Yaskawa INFORM job: A_NAIHAN_0617_1_PAINT_0.JBI

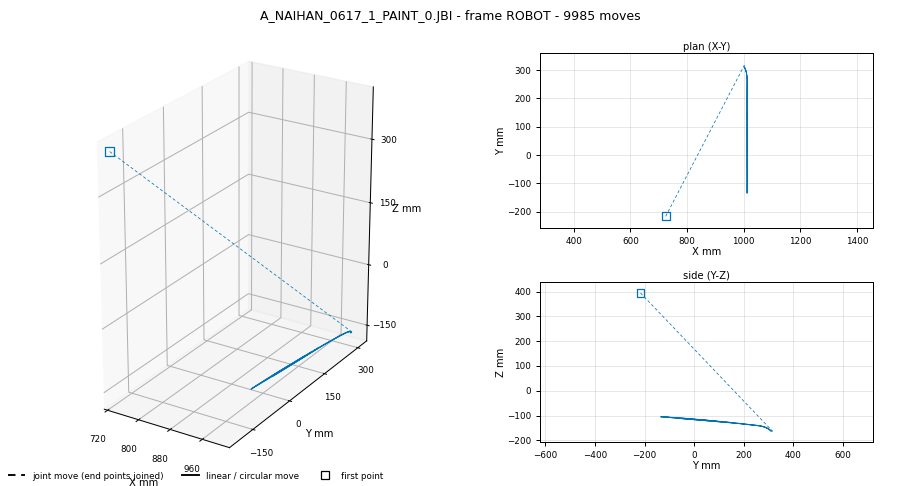
[picture p0: tool path of A_NAIHAN_0617_1_PAINT_0.JBI in frame ROBOT, 9985 of 9985 moves have a stored position in this frame; points joined in program order, loops and branches not executed]
/JOB
//NAME A_NAIHAN_0617_1_PAINT
//POS
///NPOS 9985,0,0,0,0,0
///TOOL 1
///USER 0
///POSTYPE ROBOT
///RECTAN
///RCONF 0,0,0,1,1,0,0,0,0,0,0,0,0,0,0,0,0,0,0,0,0,0,0,0
C00000=724.889,-216.680,394.500,-180.000,-0.000,-0.000
///USER 0
///POSTYPE ROBOT
///RECTAN
///RCONF 0,0,0,0,1,0,0,0,0,0,0,0,0,0,0,0,0,0,0,0,0,0,0,0
C00001=1002.338,316.145,-163.308,164.727,56.498,159.874
///RCONF 0,0,0,0,0,0,0,0,0,0,0,0,0,0,0,0,0,0,0,0,0,0,0,0
C00002=1002.509,311.597,-162.786,164.727,56.498,159.874
C00003=1002.600,311.455,-162.633,164.739,56.513,159.880
C00004=1002.691,311.313,-162.481,164.769,56.519,159.889
C00005=1002.780,311.170,-162.330,164.773,56.536,159.893
C00006=1002.870,311.027,-162.180,164.796,56.545,159.900
C00007=1002.958,310.884,-162.030,164.807,56.560,159.905
///RCONF 0,0,0,0,1,0,0,0,0,0,0,0,0,0,0,0,0,0,0,0,0,0,0,0
C00008=1003.047,310.739,-161.880,164.829,56.569,159.913
C00009=1003.134,310.594,-161.732,164.840,56.583,159.918
C00010=1003.223,310.448,-161.584,164.859,56.594,159.925
C00011=1003.316,310.290,-161.426,164.859,56.615,159.929
C00012=1003.408,310.133,-161.268,164.882,56.624,159.936
C00013=1003.501,309.974,-161.112,164.908,56.633,159.945
C00014=1003.593,309.816,-160.955,164.920,56.648,159.950
C00015=1003.685,309.656,-160.799,164.944,56.657,159.958
C00016=1003.776,309.495,-160.644,164.961,56.670,159.965
C00017=1003.866,309.334,-160.491,164.971,56.686,159.970
C00018=1003.955,309.172,-160.337,164.989,56.698,159.977
C00019=1004.045,309.010,-160.184,165.011,56.708,159.985
C00020=1004.134,308.846,-160.032,165.021,56.724,159.990
C00021=1004.222,308.683,-159.880,165.052,56.729,159.999
C00022=1004.309,308.518,-159.730,165.058,56.748,160.004
C00023=1004.397,308.353,-159.580,165.080,56.756,160.011
C00024=1004.483,308.187,-159.431,165.098,56.769,160.018
C00025=1004.570,308.021,-159.282,165.117,56.779,160.025
C00026=1004.655,307.854,-159.134,165.136,56.789,160.032
C00027=1004.740,307.686,-158.987,165.156,56.800,160.039
C00028=1004.824,307.519,-158.840,165.173,56.811,160.045
C00029=1004.908,307.350,-158.694,165.196,56.820,160.053
C00030=1004.992,307.180,-158.550,165.212,56.832,160.059
C00031=1005.074,307.011,-158.406,165.221,56.847,160.064
C00032=1005.156,306.840,-158.262,165.239,56.858,160.071
C00033=1005.238,306.669,-158.118,165.265,56.864,160.079
C00034=1005.319,306.498,-157.977,165.281,56.875,160.085
C00035=1005.400,306.326,-157.836,165.301,56.884,160.092
C00036=1005.480,306.153,-157.694,165.323,56.892,160.099
C00037=1005.559,305.980,-157.555,165.333,56.907,160.105
C00038=1005.638,305.807,-157.416,165.360,56.911,160.112
C00039=1005.716,305.632,-157.278,165.370,56.926,160.118
C00040=1005.794,305.458,-157.139,165.395,56.930,160.125
C00041=1005.872,305.282,-157.003,165.403,56.946,160.131
C00042=1005.948,305.106,-156.867,165.426,56.953,160.138
C00043=1006.025,304.930,-156.731,165.446,56.962,160.144
C00044=1006.100,304.753,-156.595,165.463,56.970,160.151
C00045=1006.175,304.576,-156.462,165.484,56.977,160.157
C00046=1006.251,304.399,-156.329,165.503,56.985,160.164
C00047=1006.324,304.220,-156.195,165.521,56.994,160.170
C00048=1006.397,304.042,-156.063,165.544,56.999,160.177
C00049=1006.471,303.863,-155.932,165.560,57.009,160.183
C00050=1006.543,303.684,-155.802,165.571,57.021,160.189
C00051=1006.614,303.503,-155.672,165.589,57.030,160.195
C00052=1006.686,303.323,-155.543,165.616,57.032,160.202
C00053=1006.757,303.142,-155.415,165.630,57.041,160.208
C00054=1006.827,302.961,-155.286,165.652,57.046,160.215
C00055=1006.897,302.780,-155.160,165.673,57.051,160.221
C00056=1006.966,302.597,-155.034,165.683,57.065,160.226
C00057=1007.035,302.415,-154.908,165.708,57.066,160.233
C00058=1007.103,302.232,-154.784,165.720,57.078,160.239
C00059=1007.171,302.049,-154.660,165.744,57.080,160.245
C00060=1007.238,301.865,-154.537,165.754,57.092,160.250
C00061=1007.305,301.681,-154.413,165.775,57.096,160.257
C00062=1007.371,301.497,-154.292,165.794,57.101,160.263
C00063=1007.436,301.312,-154.170,165.812,57.107,160.269
C00064=1007.502,301.126,-154.050,165.831,57.112,160.275
C00065=1007.566,300.942,-153.930,165.849,57.117,160.281
C00066=1007.630,300.755,-153.811,165.867,57.123,160.286
C00067=1007.695,300.570,-153.692,165.889,57.125,160.292
C00068=1007.757,300.383,-153.574,165.904,57.132,160.298
C00069=1007.820,300.196,-153.457,165.918,57.142,160.304
C00070=1007.882,300.008,-153.341,165.934,57.148,160.309
C00071=1007.943,299.821,-153.225,165.958,57.147,160.315
C00072=1008.005,299.633,-153.110,165.972,57.155,160.321
C00073=1008.065,299.445,-152.996,165.990,57.159,160.326
C00074=1008.125,299.256,-152.882,166.000,57.170,160.331
C00075=1008.185,299.067,-152.769,166.023,57.169,160.337
C00076=1008.244,298.879,-152.656,166.039,57.175,160.342
C00077=1008.303,298.688,-152.545,166.054,57.182,160.348
C00078=1008.361,298.499,-152.433,166.078,57.178,160.353
C00079=1008.419,298.309,-152.323,166.091,57.187,160.358
C00080=1008.476,298.119,-152.213,166.109,57.189,160.364
C00081=1008.533,297.929,-152.104,166.128,57.192,160.369
C00082=1008.589,297.737,-151.995,166.143,57.196,160.374
C00083=1008.646,297.546,-151.888,166.162,57.197,160.379
C00084=1008.701,297.355,-151.780,166.178,57.201,160.385
C00085=1008.756,297.163,-151.673,166.196,57.205,160.390
C00086=1008.810,296.971,-151.567,166.215,57.205,160.395
C00087=1008.864,296.779,-151.462,166.223,57.218,160.400
C00088=1008.918,296.587,-151.358,166.240,57.220,160.405
C00089=1008.972,296.394,-151.253,166.263,57.216,160.410
C00090=1009.024,296.201,-151.150,166.275,57.224,160.415
C00091=1009.076,296.008,-151.047,166.297,57.221,160.420
C00092=1009.128,295.815,-150.945,166.310,57.227,160.425
C00093=1009.179,295.620,-150.843,166.324,57.232,160.429
C00094=1009.230,295.427,-150.742,166.339,57.236,160.434
C00095=1009.280,295.233,-150.641,166.359,57.234,160.439
C00096=1009.331,295.038,-150.542,166.369,57.242,160.444
C00097=1009.380,294.844,-150.442,166.389,57.240,160.448
C00098=1009.430,294.649,-150.344,166.401,57.247,160.453
C00099=1009.479,294.454,-150.245,166.418,57.248,160.458
C00100=1009.527,294.260,-150.148,166.434,57.249,160.462
C00101=1009.575,294.063,-150.052,166.448,57.253,160.467
C00102=1009.623,293.868,-149.955,166.465,57.253,160.471
C00103=1009.669,293.672,-149.859,166.479,57.257,160.476
C00104=1009.716,293.476,-149.764,166.492,57.263,160.481
C00105=1009.762,293.280,-149.669,166.501,57.272,160.485
C00106=1009.808,293.083,-149.575,166.520,57.270,160.489
C00107=1009.854,292.886,-149.481,166.538,57.266,160.494
C00108=1009.898,292.690,-149.389,166.550,57.273,160.498
C00109=1009.944,292.493,-149.296,166.570,57.269,160.503
C00110=1009.988,292.295,-149.204,166.581,57.274,160.507
C00111=1010.032,292.098,-149.113,166.597,57.275,160.511
C00112=1010.076,291.900,-149.022,166.606,57.284,160.515
C00113=1010.119,291.703,-148.932,166.623,57.283,160.520
C00114=1010.162,291.505,-148.842,166.636,57.284,160.524
C00115=1010.204,291.307,-148.753,166.648,57.291,160.528
C00116=1010.246,291.109,-148.664,166.666,57.288,160.532
C00117=1010.288,290.911,-148.576,166.677,57.293,160.536
C00118=1010.329,290.712,-148.489,166.691,57.295,160.540
C00119=1010.370,290.513,-148.402,166.706,57.294,160.544
C00120=1010.410,290.314,-148.315,166.719,57.299,160.549
C00121=1010.450,290.116,-148.228,166.734,57.298,160.553
C00122=1010.490,289.916,-148.144,166.746,57.302,160.557
C00123=1010.530,289.717,-148.058,166.758,57.307,160.561
C00124=1010.569,289.517,-147.974,166.766,57.315,160.565
C00125=1010.607,289.318,-147.890,166.782,57.314,160.569
C00126=1010.646,289.118,-147.806,166.799,57.310,160.572
C00127=1010.684,288.918,-147.723,166.809,57.316,160.577
C00128=1010.721,288.719,-147.640,166.825,57.312,160.580
C00129=1010.758,288.519,-147.559,166.831,57.325,160.584
C00130=1010.795,288.318,-147.478,166.841,57.331,160.588
C00131=1010.832,288.117,-147.396,166.858,57.327,160.592
C00132=1010.868,287.917,-147.315,166.874,57.324,160.596
C00133=1010.904,287.716,-147.235,166.881,57.335,160.600
C00134=1010.940,287.515,-147.156,166.892,57.337,160.603
C00135=1010.975,287.314,-147.076,166.911,57.329,160.606
C00136=1011.010,287.114,-146.997,166.922,57.332,160.610
C00137=1011.044,286.913,-146.919,166.934,57.333,160.614
C00138=1011.078,286.712,-146.841,166.948,57.333,160.617
C00139=1011.113,286.510,-146.764,166.959,57.336,160.621
C00140=1011.146,286.309,-146.687,166.971,57.337,160.625
C00141=1011.179,286.107,-146.611,166.977,57.348,160.628
C00142=1011.212,285.906,-146.535,166.988,57.350,160.632
C00143=1011.244,285.704,-146.460,167.005,57.343,160.635
C00144=1011.276,285.502,-146.384,167.016,57.345,160.638
C00145=1011.309,285.300,-146.310,167.026,57.349,160.642
C00146=1011.341,285.098,-146.235,167.042,57.343,160.645
C00147=1011.371,284.896,-146.162,167.051,57.348,160.648
C00148=1011.402,284.693,-146.088,167.065,57.346,160.652
C00149=1011.433,284.491,-146.017,167.072,57.355,160.655
C00150=1011.463,284.288,-145.943,167.082,57.358,160.659
C00151=1011.494,284.086,-145.872,167.097,57.352,160.661
C00152=1011.523,283.883,-145.800,167.106,57.358,160.665
C00153=1011.552,283.680,-145.729,167.116,57.361,160.669
C00154=1011.582,283.478,-145.658,167.131,57.356,160.671
C00155=1011.610,283.275,-145.588,167.141,57.359,160.675
C00156=1011.639,283.072,-145.519,167.152,57.360,160.678
C00157=1011.666,282.868,-145.449,167.164,57.359,160.681
C00158=1011.694,282.665,-145.381,167.174,57.362,160.684
C00159=1011.722,282.462,-145.312,167.185,57.362,160.687
C00160=1011.749,282.258,-145.245,167.192,57.373,160.691
C00161=1011.776,282.054,-145.178,167.201,57.375,160.694
C00162=1011.802,281.851,-145.110,167.216,57.368,160.697
C00163=1011.829,281.648,-145.043,167.226,57.369,160.700
C00164=1011.855,281.444,-144.977,167.235,57.373,160.703
C00165=1011.880,281.240,-144.911,167.250,57.368,160.706
C00166=1011.906,281.036,-144.846,167.255,57.379,160.710
C00167=1011.931,280.832,-144.781,167.263,57.386,160.713
C00168=1011.956,280.627,-144.716,167.274,57.385,160.716
C00169=1011.981,280.424,-144.652,167.290,57.375,160.718
C00170=1012.005,280.220,-144.588,167.296,57.383,160.722
C00171=1012.028,280.015,-144.524,167.303,57.391,160.725
C00172=1012.052,279.811,-144.462,167.314,57.391,160.728
C00173=1012.076,279.607,-144.399,167.329,57.381,160.730
C00174=1012.099,279.402,-144.336,167.339,57.381,160.733
C00175=1012.122,279.197,-144.274,167.349,57.383,160.736
C00176=1012.145,278.993,-144.213,167.360,57.384,160.739
C00177=1012.166,278.788,-144.153,167.365,57.396,160.743
C00178=1012.188,278.583,-144.093,167.373,57.401,160.746
C00179=1012.210,278.378,-144.032,167.386,57.396,160.749
C00180=1012.232,278.174,-143.972,167.400,57.386,160.750
C00181=1012.252,277.969,-143.912,167.406,57.396,160.754
C00182=1012.273,277.764,-143.853,167.415,57.397,160.757
C00183=1012.294,277.559,-143.794,167.429,57.389,160.759
C00184=1012.314,277.353,-143.737,167.436,57.397,160.763
C00185=1012.334,277.149,-143.679,167.447,57.396,160.765
C00186=1012.353,276.943,-143.622,167.455,57.401,160.769
C00187=1012.373,276.738,-143.565,167.462,57.409,160.772
C00188=1012.392,276.533,-143.508,167.472,57.407,160.775
C00189=1012.412,276.327,-143.452,167.485,57.401,160.777
C00190=1012.429,276.121,-143.396,167.491,57.412,160.781
C00191=1012.448,275.916,-143.341,167.500,57.415,160.784
C00192=1012.466,275.711,-143.285,167.512,57.410,160.786
C00193=1012.483,275.505,-143.231,167.522,57.412,160.789
C00194=1012.501,275.300,-143.177,167.530,57.414,160.792
C00195=1012.518,275.094,-143.123,167.540,57.414,160.794
C00196=1012.535,274.888,-143.070,167.545,57.427,160.799
C00197=1012.552,274.682,-143.017,167.553,57.433,160.802
C00198=1012.568,274.477,-142.964,167.564,57.430,160.804
C00199=1012.585,274.270,-142.911,167.577,57.420,160.806
C00200=1012.600,274.064,-142.859,167.583,57.430,160.810
C00201=1012.616,273.858,-142.807,167.593,57.433,160.813
C00202=1012.631,273.652,-142.756,167.604,57.428,160.815
C00203=1012.645,273.446,-142.706,167.609,57.444,160.820
C00204=1012.660,273.240,-142.656,167.615,57.454,160.823
C00205=1012.676,273.033,-142.606,167.624,57.456,160.826
C00206=1012.689,272.827,-142.556,167.636,57.450,160.828
C00207=1012.704,272.621,-142.507,167.646,57.444,160.830
C00208=1012.717,272.414,-142.458,167.652,57.460,160.835
C00209=1012.730,272.208,-142.409,167.658,57.468,160.838
C00210=1012.744,272.002,-142.361,167.668,57.468,160.841
C00211=1012.756,271.795,-142.313,167.681,57.459,160.843
C00212=1012.769,271.588,-142.266,167.689,57.465,160.846
C00213=1012.781,271.382,-142.219,167.695,57.478,160.851
C00214=1012.794,271.175,-142.172,167.701,57.484,160.854
C00215=1012.805,270.969,-142.126,167.712,57.482,160.856
C00216=1012.817,270.762,-142.079,167.724,57.471,160.857
C00217=1012.828,270.555,-142.033,167.731,57.480,160.861
C00218=1012.839,270.349,-141.989,167.738,57.488,160.865
C00219=1012.850,270.142,-141.944,167.748,57.487,160.867
C00220=1012.861,269.935,-141.900,167.757,57.487,160.869
C00221=1012.871,269.729,-141.856,167.761,57.507,160.875
C00222=1012.880,269.521,-141.813,167.768,57.518,160.879
C00223=1012.900,269.107,-141.726,167.786,57.518,160.884
C00224=1012.919,268.693,-141.641,167.803,57.523,160.890
C00225=1012.935,268.278,-141.559,167.817,57.545,160.899
C00226=1012.952,267.864,-141.476,167.837,57.534,160.902
C00227=1012.967,267.450,-141.396,167.851,57.554,160.910
C00228=1012.980,267.035,-141.317,167.867,57.562,160.916
C00229=1012.994,266.620,-141.239,167.885,57.562,160.921
C00230=1013.006,266.205,-141.163,167.900,57.573,160.928
C00231=1013.017,265.790,-141.088,167.914,57.596,160.937
C00232=1013.026,265.375,-141.016,167.928,57.615,160.945
C00233=1013.036,264.960,-140.943,167.947,57.602,160.947
C00234=1013.043,264.544,-140.874,167.959,57.637,160.959
C00235=1013.050,264.128,-140.805,167.974,57.647,160.965
C00236=1013.057,263.713,-140.738,167.991,57.644,160.969
C00237=1013.061,263.297,-140.672,168.004,57.673,160.979
C00238=1013.066,262.881,-140.607,168.021,57.668,160.983
C00239=1013.069,262.465,-140.544,168.035,57.690,160.992
C00240=1013.070,262.050,-140.482,168.051,57.695,160.997
C00241=1013.071,261.634,-140.423,168.062,57.735,161.009
C00242=1013.071,261.217,-140.364,168.077,57.743,161.015
C00243=1013.070,260.801,-140.307,168.091,57.753,161.022
C00244=1013.068,260.385,-140.252,168.104,57.784,161.032
C00245=1013.065,259.969,-140.197,168.120,57.783,161.036
C00246=1013.051,258.709,-140.041,168.162,57.825,161.058
C00247=1013.047,258.464,-140.011,168.156,57.833,161.058
C00248=1013.043,258.219,-139.982,168.151,57.841,161.059
C00249=1013.039,257.973,-139.953,168.146,57.849,161.059
C00250=1013.036,257.728,-139.924,168.142,57.858,161.060
C00251=1013.032,257.482,-139.895,168.137,57.865,161.060
C00252=1013.028,257.237,-139.866,168.132,57.873,161.061
C00253=1013.024,256.992,-139.837,168.127,57.881,161.061
C00254=1013.021,256.747,-139.808,168.122,57.888,161.061
C00255=1013.017,256.502,-139.779,168.118,57.895,161.062
C00256=1013.013,256.256,-139.750,168.113,57.903,161.062
C00257=1013.009,256.011,-139.722,168.109,57.910,161.063
C00258=1013.005,255.766,-139.692,168.103,57.919,161.063
C00259=1013.002,255.521,-139.663,168.099,57.927,161.064
C00260=1012.998,255.276,-139.635,168.093,57.935,161.064
C00261=1012.995,255.030,-139.606,168.089,57.944,161.065
C00262=1012.991,254.785,-139.577,168.085,57.951,161.066
C00263=1012.987,254.539,-139.548,168.079,57.959,161.066
C00264=1012.984,254.294,-139.519,168.075,57.966,161.067
C00265=1012.980,254.049,-139.490,168.070,57.974,161.067
C00266=1012.976,253.803,-139.461,168.065,57.982,161.067
C00267=1012.973,253.558,-139.432,168.061,57.989,161.068
C00268=1012.970,253.313,-139.404,168.056,57.997,161.069
C00269=1012.966,253.067,-139.375,168.051,58.006,161.069
C00270=1012.962,252.822,-139.346,168.046,58.013,161.070
C00271=1012.958,252.577,-139.317,168.041,58.023,161.070
C00272=1012.954,252.331,-139.289,168.037,58.030,161.071
C00273=1012.951,252.086,-139.260,168.032,58.038,161.071
C00274=1012.948,251.841,-139.231,168.028,58.046,161.072
C00275=1012.945,251.596,-139.203,168.023,58.054,161.073
C00276=1012.941,251.350,-139.174,168.018,58.061,161.073
C00277=1012.937,251.105,-139.145,168.014,58.069,161.073
C00278=1012.934,250.859,-139.117,168.008,58.076,161.074
C00279=1012.930,250.614,-139.087,168.004,58.085,161.074
C00280=1012.927,250.369,-139.059,167.999,58.093,161.075
C00281=1012.923,250.123,-139.031,167.994,58.102,161.076
C00282=1012.919,249.878,-139.002,167.990,58.110,161.076
C00283=1012.916,249.632,-138.974,167.985,58.118,161.077
C00284=1012.912,249.387,-138.945,167.980,58.126,161.077
C00285=1012.909,249.142,-138.916,167.975,58.134,161.078
C00286=1012.906,248.897,-138.888,167.971,58.142,161.078
C00287=1012.902,248.652,-138.859,167.966,58.150,161.079
C00288=1012.898,248.405,-138.830,167.962,58.158,161.079
C00289=1012.895,248.160,-138.801,167.956,58.165,161.080
C00290=1012.892,247.915,-138.773,167.953,58.174,161.081
C00291=1012.888,247.670,-138.745,167.948,58.183,161.081
C00292=1012.885,247.424,-138.717,167.943,58.191,161.082
C00293=1012.881,247.178,-138.688,167.938,58.200,161.083
C00294=1012.877,246.933,-138.659,167.934,58.208,161.083
C00295=1012.874,246.688,-138.631,167.929,58.216,161.084
C00296=1012.871,246.443,-138.602,167.925,58.224,161.084
C00297=1012.868,246.197,-138.574,167.920,58.232,161.085
C00298=1012.864,245.952,-138.545,167.916,58.239,161.085
C00299=1012.861,245.706,-138.517,167.911,58.247,161.086
C00300=1012.857,245.460,-138.489,167.906,58.256,161.086
C00301=1012.853,245.215,-138.460,167.902,58.264,161.087
C00302=1012.850,244.970,-138.432,167.897,58.273,161.088
C00303=1012.847,244.724,-138.404,167.893,58.281,161.088
C00304=1012.844,244.479,-138.375,167.888,58.290,161.089
C00305=1012.841,244.234,-138.347,167.883,58.298,161.090
C00306=1012.838,243.988,-138.319,167.879,58.306,161.090
C00307=1012.834,243.742,-138.290,167.874,58.314,161.091
C00308=1012.830,243.497,-138.262,167.870,58.322,161.091
C00309=1012.827,243.251,-138.234,167.865,58.330,161.092
C00310=1012.823,243.006,-138.205,167.861,58.338,161.093
C00311=1012.820,242.760,-138.177,167.856,58.347,161.093
C00312=1012.817,242.515,-138.148,167.852,58.356,161.094
C00313=1012.814,242.270,-138.120,167.847,58.364,161.094
C00314=1012.811,242.024,-138.092,167.843,58.373,161.095
C00315=1012.808,241.779,-138.064,167.838,58.382,161.096
C00316=1012.804,241.533,-138.036,167.833,58.390,161.097
C00317=1012.801,241.288,-138.008,167.829,58.398,161.097
C00318=1012.797,241.043,-137.979,167.824,58.407,161.098
C00319=1012.794,240.797,-137.951,167.820,58.415,161.098
C00320=1012.791,240.551,-137.923,167.815,58.423,161.099
C00321=1012.788,240.306,-137.895,167.811,58.431,161.100
C00322=1012.785,240.060,-137.867,167.807,58.439,161.100
C00323=1012.782,239.815,-137.838,167.802,58.448,161.101
C00324=1012.779,239.569,-137.810,167.798,58.456,161.102
C00325=1012.775,239.324,-137.783,167.793,58.465,161.102
C00326=1012.772,239.078,-137.754,167.789,58.474,161.103
C00327=1012.768,238.833,-137.726,167.783,58.482,161.104
C00328=1012.765,238.587,-137.698,167.780,58.491,161.105
C00329=1012.762,238.341,-137.670,167.775,58.499,161.105
C00330=1012.759,238.096,-137.642,167.771,58.507,161.106
C00331=1012.756,237.850,-137.614,167.767,58.516,161.107
C00332=1012.753,237.605,-137.585,167.762,58.524,161.107
C00333=1012.749,237.359,-137.558,167.758,58.533,161.108
C00334=1012.746,237.114,-137.530,167.753,58.542,161.109
C00335=1012.743,236.868,-137.502,167.749,58.551,161.109
C00336=1012.740,236.623,-137.473,167.743,58.559,161.110
C00337=1012.737,236.377,-137.445,167.740,58.568,161.111
C00338=1012.733,236.131,-137.417,167.735,58.577,161.111
C00339=1012.731,235.885,-137.390,167.730,58.585,161.112
C00340=1012.727,235.640,-137.362,167.727,58.593,161.113
C00341=1012.724,235.394,-137.334,167.722,58.601,161.113
C00342=1012.721,235.149,-137.306,167.718,58.609,161.114
C00343=1012.718,234.904,-137.278,167.713,58.618,161.115
C00344=1012.715,234.658,-137.250,167.709,58.627,161.116
C00345=1012.712,234.412,-137.222,167.704,58.636,161.116
C00346=1012.709,234.166,-137.194,167.700,58.645,161.117
C00347=1012.706,233.921,-137.166,167.696,58.654,161.118
C00348=1012.702,233.675,-137.138,167.692,58.663,161.119
C00349=1012.699,233.429,-137.111,167.686,58.671,161.119
C00350=1012.696,233.184,-137.083,167.682,58.680,161.120
C00351=1012.694,232.939,-137.055,167.678,58.688,161.121
C00352=1012.690,232.693,-137.027,167.674,58.697,161.121
C00353=1012.688,232.447,-136.999,167.670,58.705,161.122
C00354=1012.685,232.201,-136.971,167.665,58.714,161.123
C00355=1012.681,231.956,-136.943,167.660,58.723,161.123
C00356=1012.678,231.710,-136.916,167.656,58.732,161.124
C00357=1012.675,231.465,-136.888,167.652,58.741,161.125
C00358=1012.672,231.219,-136.860,167.648,58.749,161.126
C00359=1012.669,230.973,-136.833,167.643,58.759,161.127
C00360=1012.666,230.727,-136.805,167.639,58.767,161.128
C00361=1012.664,230.481,-136.777,167.635,58.776,161.128
C00362=1012.660,230.236,-136.749,167.630,58.784,161.129
///RCONF 0,0,0,0,0,0,0,0,0,0,0,0,0,0,0,0,0,0,0,0,0,0,0,0
C00363=1012.658,229.991,-136.721,167.626,58.793,161.130
C00364=1012.654,229.745,-136.694,167.622,58.801,161.130
C00365=1012.651,229.499,-136.666,167.617,58.810,161.131
C00366=1012.648,229.253,-136.639,167.614,58.820,161.132
C00367=1012.646,229.008,-136.611,167.609,58.829,161.133
C00368=1012.643,228.762,-136.583,167.604,58.838,161.134
C00369=1012.640,228.516,-136.555,167.600,58.847,161.134
C00370=1012.637,228.270,-136.528,167.596,58.856,161.135
C00371=1012.634,228.024,-136.500,167.592,58.865,161.136
C00372=1012.631,227.779,-136.473,167.588,58.873,161.137
C00373=1012.628,227.534,-136.445,167.583,58.882,161.137
C00374=1012.625,227.287,-136.417,167.579,58.891,161.138
C00375=1012.622,227.042,-136.389,167.575,58.899,161.139
C00376=1012.620,226.796,-136.362,167.570,58.908,161.140
C00377=1012.617,226.551,-136.334,167.566,58.918,161.140
C00378=1012.614,226.305,-136.307,167.562,58.926,161.141
C00379=1012.612,226.059,-136.280,167.558,58.936,161.142
C00380=1012.608,225.814,-136.252,167.554,58.945,161.143
C00381=1012.605,225.567,-136.224,167.549,58.954,161.144
C00382=1012.602,225.321,-136.197,167.545,58.963,161.145
C00383=1012.600,225.076,-136.169,167.541,58.971,161.145
C00384=1012.597,224.830,-136.142,167.536,58.980,161.146
C00385=1012.594,224.585,-136.114,167.533,58.989,161.147
C00386=1012.592,224.339,-136.087,167.529,58.998,161.148
C00387=1012.589,224.093,-136.059,167.524,59.007,161.149
C00388=1012.585,223.847,-136.032,167.520,59.017,161.150
C00389=1012.583,223.602,-136.004,167.515,59.026,161.150
C00390=1012.580,223.356,-135.977,167.511,59.035,161.151
C00391=1012.577,223.110,-135.949,167.507,59.044,161.152
C00392=1012.575,222.864,-135.922,167.503,59.053,161.153
C00393=1012.572,222.618,-135.894,167.498,59.062,161.154
C00394=1012.569,222.372,-135.867,167.494,59.070,161.154
C00395=1012.567,222.127,-135.840,167.491,59.079,161.155
C00396=1012.564,221.880,-135.812,167.486,59.088,161.156
C00397=1012.561,221.634,-135.785,167.482,59.097,161.157
C00398=1012.558,221.390,-135.758,167.477,59.106,161.158
C00399=1012.555,221.143,-135.730,167.474,59.116,161.159
C00400=1012.553,220.898,-135.703,167.470,59.125,161.160
C00401=1012.550,220.652,-135.676,167.466,59.134,161.160
C00402=1012.548,220.402,-135.648,167.461,59.143,161.161
C00403=1012.545,220.142,-135.618,167.457,59.153,161.162
C00404=1012.541,219.869,-135.589,167.453,59.163,161.163
C00405=1012.538,219.589,-135.558,167.448,59.173,161.164
C00406=1012.535,219.292,-135.524,167.443,59.184,161.165
C00407=1012.533,218.989,-135.491,167.438,59.196,161.166
C00408=1012.529,218.693,-135.458,167.433,59.207,161.168
C00409=1012.526,218.399,-135.425,167.427,59.218,161.168
C00410=1012.523,218.110,-135.394,167.423,59.229,161.169
C00411=1012.520,217.830,-135.362,167.419,59.239,161.170
C00412=1012.517,217.564,-135.333,167.414,59.250,161.171
C00413=1012.514,217.305,-135.304,167.409,59.260,161.172
C00414=1012.511,217.050,-135.276,167.405,59.269,161.173
C00415=1012.508,216.802,-135.248,167.402,59.278,161.174
C00416=1012.506,216.556,-135.221,167.397,59.287,161.175
C00417=1012.503,216.310,-135.193,167.393,59.297,161.176
C00418=1012.501,216.065,-135.166,167.389,59.306,161.177
C00419=1012.498,215.819,-135.140,167.384,59.315,161.178
C00420=1012.495,215.573,-135.112,167.381,59.325,161.179
C00421=1012.493,215.328,-135.085,167.377,59.334,161.180
C00422=1012.491,215.084,-135.059,167.373,59.343,161.180
C00423=1012.488,214.838,-135.031,167.369,59.353,161.181
C00424=1012.485,214.593,-135.005,167.364,59.362,161.182
C00425=1012.483,214.349,-134.978,167.361,59.371,161.183
C00426=1012.480,214.104,-134.950,167.357,59.381,161.184
C00427=1012.479,213.860,-134.924,167.353,59.390,161.185
C00428=1012.476,213.616,-134.897,167.349,59.400,161.186
C00429=1012.473,213.372,-134.870,167.345,59.409,161.187
C00430=1012.471,213.128,-134.843,167.340,59.418,161.188
C00431=1012.469,212.885,-134.817,167.337,59.427,161.189
C00432=1012.466,212.642,-134.789,167.333,59.437,161.190
C00433=1012.464,212.398,-134.763,167.329,59.447,161.191
C00434=1012.461,212.155,-134.736,167.325,59.455,161.192
C00435=1012.459,211.911,-134.709,167.320,59.465,161.192
C00436=1012.456,211.669,-134.683,167.317,59.474,161.194
C00437=1012.454,211.426,-134.656,167.313,59.483,161.194
C00438=1012.451,211.184,-134.629,167.310,59.493,161.195
C00439=1012.449,210.941,-134.603,167.305,59.502,161.196
C00440=1012.446,210.698,-134.576,167.302,59.512,161.197
C00441=1012.444,210.456,-134.549,167.297,59.521,161.198
C00442=1012.442,210.214,-134.523,167.293,59.531,161.199
C00443=1012.439,209.971,-134.496,167.290,59.540,161.200
C00444=1012.437,209.728,-134.470,167.286,59.550,161.201
C00445=1012.434,209.486,-134.443,167.282,59.559,161.202
C00446=1012.433,209.243,-134.417,167.278,59.569,161.203
C00447=1012.430,209.001,-134.390,167.274,59.577,161.204
C00448=1012.427,208.758,-134.363,167.270,59.587,161.205
C00449=1012.425,208.515,-134.337,167.267,59.596,161.206
C00450=1012.423,208.274,-134.310,167.262,59.606,161.207
C00451=1012.421,208.031,-134.284,167.259,59.615,161.208
C00452=1012.418,207.788,-134.257,167.255,59.625,161.209
C00453=1012.415,207.545,-134.231,167.250,59.634,161.210
C00454=1012.413,207.302,-134.204,167.247,59.644,161.211
C00455=1012.411,207.059,-134.178,167.243,59.653,161.212
C00456=1012.409,206.816,-134.151,167.240,59.663,161.213
C00457=1012.407,206.572,-134.125,167.235,59.672,161.214
C00458=1012.405,206.329,-134.098,167.231,59.682,161.215
C00459=1012.402,206.086,-134.072,167.228,59.692,161.216
C00460=1012.400,205.842,-134.045,167.223,59.701,161.217
C00461=1012.397,205.598,-134.018,167.221,59.711,161.218
C00462=1012.395,205.354,-133.992,167.217,59.721,161.219
C00463=1012.393,205.110,-133.965,167.212,59.730,161.220
C00464=1012.390,204.866,-133.939,167.209,59.739,161.221
C00465=1012.388,204.622,-133.912,167.205,59.749,161.222
C00466=1012.386,204.377,-133.886,167.200,59.759,161.223
C00467=1012.384,204.134,-133.859,167.197,59.768,161.224
C00468=1012.381,203.891,-133.833,167.193,59.778,161.225
C00469=1012.379,203.646,-133.806,167.189,59.788,161.226
C00470=1012.373,202.396,-133.669,166.565,59.695,161.014
C00471=1012.373,202.178,-133.645,166.562,59.705,161.015
C00472=1012.373,201.767,-133.601,166.555,59.722,161.017
C00473=1012.373,201.556,-133.577,166.553,59.730,161.018
C00474=1012.373,201.338,-133.555,166.549,59.739,161.019
C00475=1012.373,201.115,-133.530,166.546,59.749,161.020
C00476=1012.373,200.877,-133.505,166.542,59.759,161.021
C00477=1012.373,200.622,-133.477,166.538,59.770,161.022
C00478=1012.373,200.367,-133.449,166.534,59.780,161.023
C00479=1012.372,200.126,-133.424,166.532,59.790,161.025
C00480=1012.373,199.893,-133.398,166.527,59.799,161.025
C00481=1012.373,199.664,-133.374,166.524,59.809,161.026
C00482=1012.373,199.422,-133.347,166.520,59.819,161.027
C00483=1012.372,199.031,-133.305,166.516,59.835,161.029
C00484=1012.373,198.640,-133.263,166.510,59.852,161.031
C00485=1012.372,198.393,-133.236,166.506,59.862,161.032
C00486=1012.372,198.157,-133.211,166.502,59.872,161.033
C00487=1012.373,197.921,-133.185,166.499,59.882,161.034
C00488=1012.372,197.685,-133.160,166.495,59.892,161.035
C00489=1012.372,197.449,-133.135,166.492,59.902,161.037
C00490=1012.373,197.213,-133.109,166.489,59.911,161.038
C00491=1012.372,196.977,-133.084,166.486,59.921,161.039
C00492=1012.372,196.741,-133.059,166.482,59.931,161.040
C00493=1012.373,196.505,-133.033,166.479,59.940,161.041
C00494=1012.373,196.269,-133.008,166.475,59.949,161.042
C00495=1012.373,196.033,-132.983,166.472,59.959,161.043
C00496=1012.372,195.797,-132.958,166.469,59.970,161.044
C00497=1012.373,195.561,-132.932,166.466,59.979,161.045
C00498=1012.373,195.325,-132.906,166.463,59.989,161.046
C00499=1012.373,195.090,-132.881,166.459,59.999,161.047
C00500=1012.372,194.853,-132.855,166.456,60.009,161.048
C00501=1012.372,194.617,-132.830,166.452,60.018,161.049
C00502=1012.373,194.381,-132.805,166.449,60.027,161.050
C00503=1012.373,194.145,-132.780,166.446,60.037,161.051
C00504=1012.373,193.910,-132.755,166.443,60.047,161.053
C00505=1012.373,193.673,-132.729,166.440,60.056,161.054
C00506=1012.372,193.437,-132.704,166.436,60.066,161.055
C00507=1012.373,193.201,-132.678,166.433,60.076,161.056
C00508=1012.373,192.965,-132.653,166.430,60.086,161.057
C00509=1012.373,192.730,-132.628,166.427,60.095,161.058
C00510=1012.374,192.493,-132.603,166.424,60.105,161.059
C00511=1012.373,192.257,-132.578,166.420,60.114,161.060
C00512=1012.374,192.021,-132.553,166.417,60.123,161.061
C00513=1012.373,191.785,-132.528,166.414,60.133,161.062
C00514=1012.374,191.549,-132.502,166.410,60.142,161.063
C00515=1012.374,191.313,-132.477,166.407,60.152,161.064
C00516=1012.374,191.078,-132.452,166.405,60.162,161.066
C00517=1012.374,190.842,-132.427,166.400,60.171,161.066
C00518=1012.374,190.606,-132.402,166.397,60.181,161.068
C00519=1012.374,190.369,-132.376,166.394,60.191,161.069
C00520=1012.374,190.134,-132.351,166.392,60.200,161.070
C00521=1012.374,189.898,-132.326,166.389,60.210,161.071
C00522=1012.375,189.662,-132.300,166.385,60.219,161.072
C00523=1012.374,189.426,-132.275,166.383,60.228,161.073
C00524=1012.375,189.189,-132.251,166.380,60.238,161.074
C00525=1012.375,188.954,-132.226,166.377,60.247,161.075
C00526=1012.375,188.718,-132.200,166.374,60.257,161.077
C00527=1012.375,188.482,-132.175,166.370,60.267,161.078
C00528=1012.376,188.246,-132.150,166.367,60.277,161.079
C00529=1012.375,188.011,-132.125,166.365,60.285,161.080
C00530=1012.376,187.775,-132.100,166.362,60.295,161.081
C00531=1012.376,187.539,-132.074,166.359,60.305,161.082
C00532=1012.376,187.302,-132.050,166.355,60.314,161.083
C00533=1012.377,187.066,-132.025,166.352,60.323,161.084
C00534=1012.377,186.831,-132.000,166.350,60.332,161.085
C00535=1012.377,186.595,-131.974,166.347,60.341,161.086
C00536=1012.377,186.359,-131.949,166.343,60.352,161.087
C00537=1012.377,186.123,-131.924,166.341,60.361,161.088
C00538=1012.377,185.887,-131.900,166.338,60.370,161.090
C00539=1012.378,185.651,-131.874,166.335,60.380,161.091
C00540=1012.378,185.415,-131.849,166.331,60.389,161.092
C00541=1012.378,185.179,-131.824,166.328,60.399,161.093
C00542=1012.378,184.944,-131.799,166.326,60.408,161.094
C00543=1012.378,184.708,-131.774,166.323,60.417,161.095
C00544=1012.378,184.471,-131.750,166.320,60.427,161.096
C00545=1012.379,184.235,-131.724,166.316,60.435,161.097
C00546=1012.379,184.000,-131.699,166.313,60.445,161.098
C00547=1012.379,183.764,-131.674,166.312,60.454,161.099
C00548=1012.379,183.528,-131.649,166.309,60.464,161.101
C00549=1012.380,183.292,-131.624,166.306,60.474,161.102
C00550=1012.380,183.056,-131.599,166.302,60.483,161.103
C00551=1012.380,182.820,-131.574,166.300,60.492,161.104
C00552=1012.381,182.585,-131.549,166.297,60.501,161.105
C00553=1012.381,182.348,-131.525,166.295,60.510,161.106
C00554=1012.381,182.112,-131.499,166.291,60.519,161.107
C00555=1012.381,181.877,-131.474,166.288,60.529,161.108
C00556=1012.381,181.641,-131.449,166.285,60.538,161.109
C00557=1012.382,181.405,-131.425,166.284,60.548,161.111
C00558=1012.381,181.169,-131.400,166.280,60.557,161.111
C00559=1012.382,180.934,-131.375,166.277,60.566,161.113
C00560=1012.382,180.698,-131.350,166.275,60.575,161.114
C00561=1012.383,180.461,-131.325,166.272,60.585,161.115
C00562=1012.383,180.226,-131.300,166.269,60.593,161.116
C00563=1012.383,179.990,-131.275,166.266,60.603,161.117
C00564=1012.383,179.754,-131.250,166.264,60.611,161.118
C00565=1012.384,179.518,-131.226,166.261,60.621,161.119
C00566=1012.384,179.283,-131.201,166.258,60.631,161.120
C00567=1012.384,179.047,-131.175,166.254,60.640,161.121
C00568=1012.385,178.810,-131.151,166.253,60.649,161.123
C00569=1012.385,178.574,-131.126,166.250,60.659,161.124
C00570=1012.385,178.339,-131.101,166.247,60.667,161.125
C00571=1012.385,178.104,-131.076,166.244,60.676,161.126
C00572=1012.386,177.867,-131.052,166.242,60.685,161.127
C00573=1012.386,177.632,-131.027,166.239,60.694,161.128
C00574=1012.387,177.396,-131.002,166.237,60.704,161.129
C00575=1012.387,177.160,-130.977,166.234,60.712,161.130
C00576=1012.387,176.924,-130.952,166.231,60.722,161.131
C00577=1012.387,176.688,-130.927,166.228,60.732,161.133
C00578=1012.388,176.453,-130.903,166.226,60.740,161.134
C00579=1012.388,176.217,-130.878,166.223,60.750,161.135
C00580=1012.388,175.981,-130.853,166.221,60.758,161.136
C00581=1012.389,175.745,-130.829,166.218,60.767,161.137
C00582=1012.389,175.510,-130.804,166.215,60.777,161.138
C00583=1012.389,175.274,-130.778,166.213,60.785,161.139
C00584=1012.390,175.038,-130.755,166.210,60.794,161.140
C00585=1012.390,174.802,-130.730,166.207,60.803,161.141
C00586=1012.390,174.566,-130.704,166.206,60.813,161.143
C00587=1012.391,174.331,-130.680,166.202,60.822,161.143
C00588=1012.391,174.095,-130.656,166.200,60.831,161.145
C00589=1012.391,173.859,-130.630,166.197,60.840,161.146
C00590=1012.392,173.624,-130.606,166.195,60.849,161.147
C00591=1012.392,173.388,-130.581,166.193,60.858,161.148
C00592=1012.392,173.151,-130.557,166.190,60.866,161.149
C00593=1012.393,172.917,-130.532,166.188,60.875,161.150
C00594=1012.393,172.681,-130.507,166.185,60.884,161.151
C00595=1012.394,172.445,-130.483,166.182,60.893,161.152
C00596=1012.393,172.209,-130.458,166.180,60.903,161.154
C00597=1012.394,171.973,-130.433,166.177,60.911,161.155
C00598=1012.395,171.738,-130.409,166.175,60.921,161.156
C00599=1012.395,171.502,-130.383,166.172,60.930,161.157
C00600=1012.396,171.266,-130.360,166.169,60.938,161.158
C00601=1012.395,171.031,-130.335,166.167,60.947,161.159
C00602=1012.396,170.795,-130.310,166.165,60.956,161.160
C00603=1012.397,170.559,-130.286,166.163,60.964,161.161
C00604=1012.396,170.323,-130.261,166.160,60.973,161.163
C00605=1012.398,170.088,-130.236,166.158,60.983,161.164
C00606=1012.397,169.852,-130.211,166.155,60.991,161.165
C00607=1012.398,169.617,-130.187,166.153,61.001,161.166
C00608=1012.398,169.380,-130.162,166.150,61.010,161.167
C00609=1012.399,169.145,-130.138,166.147,61.018,161.168
C00610=1012.399,168.909,-130.114,166.145,61.027,161.169
C00611=1012.400,168.674,-130.088,166.143,61.035,161.170
C00612=1012.400,168.438,-130.064,166.141,61.045,161.172
C00613=1012.400,168.203,-130.040,166.138,61.053,161.173
C00614=1012.401,167.967,-130.014,166.136,61.062,161.174
C00615=1012.401,167.731,-129.991,166.134,61.071,161.175
C00616=1012.402,167.496,-129.966,166.131,61.080,161.176
C00617=1012.402,167.260,-129.942,166.128,61.089,161.177
C00618=1012.403,167.025,-129.917,166.127,61.098,161.178
C00619=1012.403,166.788,-129.893,166.124,61.106,161.179
C00620=1012.403,166.553,-129.868,166.122,61.115,161.181
C00621=1012.404,166.317,-129.843,166.119,61.124,161.182
C00622=1012.404,166.082,-129.819,166.117,61.132,161.183
C00623=1012.405,165.847,-129.794,166.115,61.141,161.184
C00624=1012.405,165.611,-129.770,166.112,61.149,161.185
C00625=1012.406,165.375,-129.745,166.110,61.158,161.186
C00626=1012.406,165.072,-129.714,166.107,61.169,161.187
C00627=1012.407,164.754,-129.681,166.104,61.181,161.189
C00628=1012.407,164.366,-129.641,166.100,61.195,161.191
C00629=1012.408,164.145,-129.617,166.099,61.203,161.192
C00630=1012.408,163.925,-129.595,166.096,61.211,161.193
C00631=1012.409,163.687,-129.570,166.093,61.220,161.194
C00632=1012.409,163.424,-129.543,166.092,61.229,161.195
C00633=1012.410,163.130,-129.513,166.089,61.240,161.197
C00634=1012.410,162.821,-129.481,166.086,61.252,161.198
C00635=1012.411,162.530,-129.451,166.083,61.262,161.199
C00636=1012.412,162.224,-129.419,166.080,61.274,161.201
C00637=1012.412,161.920,-129.388,166.077,61.285,161.202
C00638=1012.413,161.628,-129.357,166.075,61.295,161.204
C00639=1012.413,161.351,-129.329,166.072,61.305,161.205
C00640=1012.414,161.088,-129.301,166.070,61.315,161.206
C00641=1012.414,160.838,-129.276,166.067,61.325,161.208
C00642=1012.414,160.597,-129.251,166.065,61.333,161.209
C00643=1012.415,160.363,-129.227,166.062,61.342,161.210
C00644=1012.416,160.132,-129.204,166.059,61.375,161.216
C00645=1012.414,159.899,-129.182,166.051,61.454,161.230
C00646=1012.412,159.664,-129.162,166.044,61.534,161.245
C00647=1012.411,159.429,-129.141,166.038,61.615,161.260
C00648=1012.410,159.192,-129.120,166.030,61.694,161.275
C00649=1012.409,158.956,-129.098,166.023,61.774,161.290
C00650=1012.408,158.722,-129.077,166.016,61.853,161.305
C00651=1012.407,158.487,-129.056,166.010,61.931,161.319
C00652=1012.406,158.250,-129.035,166.003,62.009,161.334
C00653=1012.405,158.013,-129.014,165.996,62.088,161.349
C00654=1012.404,157.775,-128.992,165.989,62.167,161.364
C00655=1012.402,157.536,-128.971,165.984,62.245,161.379
C00656=1012.401,157.298,-128.950,165.977,62.323,161.393
C00657=1012.400,157.082,-128.930,165.972,62.393,161.407
C00658=1012.399,156.819,-128.907,165.966,62.478,161.423
C00659=1012.398,156.579,-128.885,165.959,62.556,161.438
C00660=1012.397,156.341,-128.864,165.953,62.632,161.452
C00661=1012.396,156.101,-128.843,165.948,62.709,161.467
C00662=1012.395,155.862,-128.821,165.942,62.785,161.482
C00663=1012.394,155.622,-128.800,165.936,62.862,161.497
C00664=1012.393,155.382,-128.778,165.930,62.937,161.511
C00665=1012.392,155.141,-128.757,165.925,63.012,161.526
C00666=1012.391,154.902,-128.735,165.920,63.088,161.541
C00667=1012.390,154.661,-128.713,165.915,63.164,161.556
C00668=1012.389,154.420,-128.692,165.909,63.238,161.570
C00669=1012.388,154.179,-128.669,165.904,63.313,161.585
C00670=1012.387,153.938,-128.648,165.900,63.388,161.600
C00671=1012.386,153.698,-128.626,165.895,63.462,161.614
C00672=1012.385,153.455,-128.604,165.890,63.536,161.629
C00673=1012.384,153.214,-128.583,165.886,63.609,161.644
C00674=1012.383,152.972,-128.561,165.882,63.683,161.659
C00675=1012.383,152.730,-128.539,165.877,63.757,161.673
C00676=1012.382,152.487,-128.518,165.872,63.830,161.688
C00677=1012.381,152.238,-128.495,165.868,63.905,161.703
C00678=1012.380,151.984,-128.472,165.863,63.981,161.718
C00679=1012.379,151.720,-128.448,165.858,64.059,161.734
C00680=1012.378,151.450,-128.423,165.854,64.140,161.750
C00681=1012.377,151.171,-128.399,165.849,64.222,161.767
C00682=1012.376,150.884,-128.373,165.846,64.307,161.785
C00683=1012.375,150.592,-128.347,165.842,64.392,161.802
C00684=1012.374,150.295,-128.320,165.838,64.478,161.820
C00685=1012.374,149.996,-128.293,165.834,64.565,161.839
C00686=1012.373,149.695,-128.265,165.830,64.652,161.857
C00687=1012.372,149.397,-128.239,165.826,64.739,161.875
C00688=1012.371,149.101,-128.211,165.824,64.824,161.893
C00689=1012.370,148.809,-128.185,165.820,64.907,161.910
C00690=1012.369,148.524,-128.159,165.817,64.988,161.928
C00691=1012.369,148.246,-128.135,165.814,65.067,161.944
C00692=1012.368,147.976,-128.109,165.812,65.143,161.961
C00693=1012.367,147.714,-128.086,165.809,65.216,161.976
C00694=1012.366,147.460,-128.063,165.806,65.287,161.991
C00695=1012.365,147.212,-128.040,165.803,65.356,162.006
C00696=1012.365,146.968,-128.018,165.801,65.423,162.021
C00697=1012.364,146.726,-127.996,165.799,65.490,162.035
C00698=1012.364,146.484,-127.975,165.797,65.556,162.050
C00699=1012.363,146.242,-127.953,165.794,65.623,162.064
C00700=1012.363,145.999,-127.931,165.793,65.689,162.079
C00701=1012.362,145.759,-127.909,165.792,65.755,162.093
C00702=1012.361,145.516,-127.887,165.790,65.820,162.108
C00703=1012.361,145.275,-127.865,165.789,65.885,162.122
C00704=1012.361,145.033,-127.843,165.786,65.950,162.136
C00705=1012.360,144.792,-127.821,165.786,66.015,162.151
C00706=1012.360,144.550,-127.799,165.784,66.079,162.165
C00707=1012.359,144.309,-127.777,165.782,66.143,162.179
C00708=1012.359,144.069,-127.756,165.781,66.207,162.194
C00709=1012.358,143.828,-127.733,165.781,66.270,162.208
C00710=1012.357,143.588,-127.712,165.780,66.333,162.223
C00711=1012.358,143.347,-127.690,165.779,66.395,162.237
C00712=1012.357,143.108,-127.669,165.778,66.458,162.251
C00713=1012.357,142.868,-127.646,165.777,66.520,162.265
C00714=1012.356,142.628,-127.624,165.778,66.582,162.280
C00715=1012.355,142.389,-127.602,165.776,66.644,162.294
C00716=1012.355,142.150,-127.581,165.776,66.705,162.308
C00717=1012.355,141.911,-127.559,165.776,66.766,162.323
C00718=1012.354,141.666,-127.537,165.775,66.828,162.337
C00719=1012.354,141.455,-127.518,165.776,66.881,162.350
C00720=1012.353,141.199,-127.495,165.775,66.945,162.365
C00721=1012.353,140.907,-127.468,165.775,67.019,162.382
C00722=1012.353,140.655,-127.445,165.775,67.081,162.397
C00723=1012.353,140.380,-127.420,165.776,67.149,162.413
C00724=1012.352,140.085,-127.393,165.776,67.222,162.431
C00725=1012.351,139.776,-127.365,165.775,67.298,162.448
C00726=1012.351,139.464,-127.336,165.777,67.374,162.467
C00727=1012.351,139.156,-127.309,165.777,67.448,162.485
C00728=1012.350,138.862,-127.281,165.778,67.519,162.503
C00729=1012.350,138.588,-127.256,165.779,67.585,162.519
C00730=1012.349,138.336,-127.233,165.780,67.645,162.534
C00731=1012.349,137.916,-127.195,165.782,67.744,162.558
C00732=1012.349,137.532,-127.160,165.782,67.834,162.580
C00733=1012.349,137.116,-127.122,165.784,67.930,162.604
C00734=1012.348,136.733,-127.087,165.786,68.019,162.626
C00735=1012.348,136.347,-127.051,165.788,68.107,162.649
C00736=1012.348,135.928,-127.013,165.791,68.201,162.673
C00737=1012.347,135.615,-126.984,165.793,68.271,162.691
C00738=1012.347,135.422,-126.966,165.794,68.314,162.702
C00739=1012.347,135.185,-126.944,165.796,68.366,162.716
C00740=1012.347,134.776,-126.907,165.799,68.455,162.739
C00741=1012.346,134.432,-126.875,165.801,68.530,162.758
C00742=1012.398,134.450,-126.756,165.735,65.950,162.115
C00743=1012.450,134.469,-126.638,165.799,63.383,161.562
C00744=1012.453,134.949,-126.677,165.811,63.164,161.518
C00745=1012.455,135.211,-126.698,165.819,63.046,161.495
C00746=1012.457,135.496,-126.721,165.827,62.918,161.470
C00747=1012.459,135.729,-126.740,165.833,62.813,161.450
C00748=1012.460,135.954,-126.759,165.839,62.712,161.430
C00749=1012.463,136.374,-126.794,165.852,62.525,161.394
C00750=1012.465,136.760,-126.825,165.864,62.354,161.361
C00751=1012.469,137.143,-126.856,165.877,62.184,161.328
C00752=1012.472,137.560,-126.891,165.890,62.000,161.294
C00753=1012.474,137.944,-126.922,165.903,61.831,161.261
C00754=1012.477,138.365,-126.958,165.918,61.648,161.227
C00755=1012.479,138.617,-126.978,165.928,61.537,161.207
C00756=1012.480,138.891,-127.001,165.937,61.418,161.184
C00757=1012.483,139.186,-127.025,165.948,61.290,161.161
C00758=1012.485,139.494,-127.051,165.959,61.157,161.136
C00759=1012.488,139.807,-127.077,165.971,61.022,161.111
C00760=1012.490,140.115,-127.102,165.983,60.889,161.087
C00761=1012.492,140.411,-127.127,165.996,60.763,161.064
C00762=1012.494,140.686,-127.150,166.007,60.645,161.043
C00763=1012.496,141.058,-127.181,166.022,60.486,161.014
C00764=1012.497,141.231,-127.195,166.029,60.412,161.001
C00765=1012.500,141.486,-127.217,166.039,60.303,160.981
C00766=1012.501,141.698,-127.235,166.048,60.214,160.965
C00767=1012.503,141.943,-127.256,166.058,60.111,160.947
C00768=1012.504,142.182,-127.275,166.069,60.009,160.929
C00769=1012.506,142.421,-127.296,166.080,59.909,160.911
C00770=1012.508,142.661,-127.315,166.090,59.808,160.893
C00771=1012.509,142.900,-127.336,166.101,59.708,160.875
C00772=1012.512,143.140,-127.356,166.111,59.607,160.857
C00773=1012.513,143.380,-127.376,166.122,59.507,160.840
C00774=1012.515,143.621,-127.396,166.133,59.407,160.822
C00775=1012.517,143.861,-127.417,166.143,59.307,160.805
C00776=1012.518,144.102,-127.437,166.155,59.206,160.787
C00777=1012.520,144.343,-127.458,166.167,59.107,160.770
C00778=1012.522,144.584,-127.478,166.178,59.007,160.753
C00779=1012.524,144.825,-127.499,166.189,58.908,160.735
C00780=1012.526,145.067,-127.519,166.201,58.808,160.718
C00781=1012.527,145.308,-127.539,166.212,58.709,160.701
C00782=1012.530,145.550,-127.560,166.224,58.610,160.684
C00783=1012.531,145.793,-127.581,166.236,58.512,160.667
C00784=1012.533,146.034,-127.602,166.248,58.413,160.650
C00785=1012.534,146.277,-127.622,166.259,58.315,160.633
C00786=1012.536,146.519,-127.643,166.272,58.217,160.616
C00787=1012.538,146.761,-127.664,166.284,58.119,160.600
C00788=1012.540,147.004,-127.684,166.296,58.021,160.583
C00789=1012.542,147.247,-127.706,166.310,57.923,160.567
C00790=1012.544,147.495,-127.727,166.322,57.824,160.550
C00791=1012.547,147.908,-127.762,166.343,57.659,160.522
C00792=1012.346,133.023,-126.745,165.812,68.825,162.836
C00793=1012.346,133.240,-126.765,165.810,68.781,162.824
C00794=1012.346,132.959,-126.739,165.813,68.839,162.840
C00795=1012.345,132.677,-126.713,165.815,68.896,162.855
C00796=1012.346,132.465,-126.694,165.817,68.939,162.866
C00797=1012.345,132.253,-126.674,165.819,68.982,162.878
C00798=1012.391,132.287,-126.570,165.730,66.672,162.281
C00799=1012.346,132.346,-126.683,165.818,68.962,162.873
C00800=1012.346,132.770,-126.722,165.815,68.877,162.850
C00801=1012.345,132.520,-126.699,165.817,68.928,162.864
C00802=1012.345,132.272,-126.676,165.819,68.978,162.877
C00803=1012.346,132.022,-126.653,165.821,69.026,162.890
C00804=1012.345,131.774,-126.630,165.824,69.076,162.904
C00805=1012.345,131.525,-126.607,165.825,69.123,162.916
C00806=1012.346,131.275,-126.584,165.828,69.172,162.930
C00807=1012.345,131.027,-126.560,165.830,69.218,162.942
C00808=1012.345,130.778,-126.538,165.833,69.265,162.955
C00809=1012.346,130.529,-126.514,165.835,69.309,162.967
C00810=1012.345,130.280,-126.491,165.839,69.355,162.980
C00811=1012.346,130.031,-126.468,165.841,69.399,162.992
C00812=1012.345,129.782,-126.444,165.843,69.442,163.004
C00813=1012.346,129.534,-126.421,165.845,69.485,163.016
C00814=1012.346,129.285,-126.398,165.848,69.527,163.028
C00815=1012.346,129.035,-126.374,165.850,69.568,163.039
C00816=1012.346,128.787,-126.351,165.852,69.608,163.050
C00817=1012.346,128.538,-126.328,165.855,69.647,163.062
C00818=1012.346,128.289,-126.304,165.857,69.685,163.072
C00819=1012.347,128.040,-126.281,165.859,69.722,163.083
C00820=1012.347,127.791,-126.257,165.862,69.757,163.093
C00821=1012.347,127.542,-126.233,165.863,69.791,163.102
C00822=1012.348,127.293,-126.210,165.866,69.824,163.112
C00823=1012.348,127.044,-126.186,165.867,69.855,163.120
C00824=1012.348,126.795,-126.162,165.869,69.884,163.129
C00825=1012.349,126.547,-126.138,165.871,69.912,163.137
C00826=1012.349,126.298,-126.114,165.872,69.936,163.144
C00827=1012.350,126.049,-126.089,165.874,69.959,163.150
C00828=1012.350,125.801,-126.066,165.875,69.979,163.156
C00829=1012.350,125.552,-126.042,165.874,69.994,163.159
C00830=1012.351,125.302,-126.017,165.875,70.007,163.163
C00831=1012.352,125.054,-125.992,165.875,70.015,163.165
C00832=1012.353,124.805,-125.967,165.874,70.015,163.165
C00833=1012.353,124.557,-125.942,165.874,70.009,163.163
C00834=1012.355,124.308,-125.916,165.870,69.991,163.157
C00835=1012.356,124.059,-125.888,165.866,69.957,163.146
C00836=1012.359,123.658,-125.841,165.852,69.820,163.104
C00837=1012.372,123.747,-125.818,165.794,69.126,162.902
C00838=1012.375,123.986,-125.831,165.780,68.894,162.838
C00839=1012.377,124.226,-125.846,165.768,68.698,162.784
C00840=1012.380,124.467,-125.861,165.759,68.519,162.736
C00841=1012.383,124.707,-125.878,165.751,68.352,162.692
C00842=1012.384,124.947,-125.895,165.744,68.194,162.650
C00843=1012.386,125.187,-125.912,165.739,68.041,162.611
C00844=1012.388,125.428,-125.929,165.734,67.894,162.573
C00845=1012.390,125.676,-125.948,165.730,67.745,162.535
C00846=1012.392,125.926,-125.966,165.725,67.600,162.499
C00847=1012.394,126.176,-125.984,165.721,67.457,162.463
C00848=1012.396,126.424,-126.003,165.718,67.318,162.428
C00849=1012.397,126.674,-126.022,165.716,67.180,162.394
C00850=1012.399,126.923,-126.041,165.714,67.044,162.362
C00851=1012.401,127.172,-126.060,165.712,66.911,162.329
C00852=1012.402,127.422,-126.079,165.711,66.778,162.298
C00853=1012.404,127.671,-126.098,165.710,66.648,162.267
C00854=1012.406,127.920,-126.117,165.711,66.519,162.237
C00855=1012.408,128.169,-126.136,165.710,66.390,162.207
C00856=1012.410,128.419,-126.156,165.710,66.263,162.177
C00857=1012.411,128.667,-126.175,165.711,66.137,162.148
C00858=1012.413,128.917,-126.194,165.711,66.011,162.120
C00859=1012.414,129.167,-126.215,165.712,65.888,162.092
C00860=1012.416,129.416,-126.234,165.714,65.764,162.064
C00861=1012.418,129.665,-126.253,165.715,65.641,162.036
C00862=1012.419,129.914,-126.273,165.718,65.519,162.009
C00863=1012.421,130.163,-126.293,165.720,65.398,161.983
C00864=1012.423,130.413,-126.312,165.723,65.277,161.956
C00865=1012.425,130.662,-126.332,165.726,65.157,161.930
C00866=1012.426,130.912,-126.352,165.730,65.038,161.905
C00867=1012.428,131.160,-126.372,165.733,64.919,161.879
C00868=1012.430,131.409,-126.391,165.736,64.800,161.854
C00869=1012.432,131.755,-126.420,165.742,64.637,161.819
C00870=1012.434,132.101,-126.447,165.747,64.474,161.785
C00871=1012.436,132.447,-126.475,165.753,64.313,161.751
C00872=1012.438,132.792,-126.503,165.761,64.151,161.718
C00873=1012.392,132.799,-126.614,165.729,66.506,162.242
C00874=1012.345,132.806,-126.726,165.813,68.870,162.848
C00875=1012.346,133.023,-126.745,165.812,68.825,162.836
C00876=1012.606,-106.829,-106.487,165.702,74.011,164.138
C00877=1012.605,-107.083,-106.471,165.709,74.034,164.148
C00878=1012.606,-107.346,-106.455,165.710,74.041,164.151
C00879=1012.605,-107.611,-106.437,165.706,74.034,164.146
C00880=1012.605,-107.879,-106.420,165.699,74.019,164.138
C00881=1012.606,-108.128,-106.403,165.691,73.997,164.128
C00882=1012.606,-108.372,-106.386,165.680,73.971,164.114
C00883=1012.607,-108.610,-106.369,165.671,73.941,164.100
C00884=1012.607,-108.840,-106.354,165.659,73.910,164.085
C00885=1012.608,-109.084,-106.336,165.646,73.872,164.067
C00886=1012.608,-109.321,-106.319,165.632,73.833,164.049
C00887=1012.608,-109.551,-106.303,165.618,73.794,164.030
C00888=1012.609,-109.782,-106.286,165.605,73.752,164.011
C00889=1012.609,-110.032,-106.268,165.589,73.704,163.989
C00890=1012.611,-110.281,-106.250,165.573,73.654,163.966
C00891=1012.611,-110.530,-106.232,165.557,73.603,163.944
C00892=1012.612,-110.779,-106.214,165.540,73.550,163.920
C00893=1012.612,-111.028,-106.195,165.522,73.495,163.895
C00894=1012.614,-111.278,-106.177,165.506,73.439,163.871
C00895=1012.614,-111.527,-106.158,165.489,73.381,163.846
C00896=1012.615,-111.777,-106.140,165.471,73.323,163.820
C00897=1012.616,-112.025,-106.122,165.454,73.262,163.795
C00898=1012.617,-112.275,-106.103,165.435,73.200,163.767
C00899=1012.617,-112.524,-106.084,165.417,73.138,163.741
C00900=1012.618,-112.774,-106.065,165.400,73.075,163.715
C00901=1012.619,-113.023,-106.047,165.381,73.010,163.687
C00902=1012.620,-113.272,-106.028,165.362,72.944,163.660
C00903=1012.621,-113.521,-106.009,165.344,72.877,163.632
C00904=1012.623,-113.771,-105.991,165.327,72.809,163.605
C00905=1012.623,-114.020,-105.972,165.308,72.741,163.577
C00906=1012.624,-114.269,-105.953,165.290,72.672,163.549
C00907=1012.625,-114.519,-105.934,165.272,72.602,163.522
C00908=1012.626,-114.768,-105.916,165.254,72.531,163.493
C00909=1012.627,-115.017,-105.897,165.236,72.459,163.466
C00910=1012.628,-115.266,-105.877,165.219,72.387,163.438
C00911=1012.629,-115.516,-105.858,165.200,72.313,163.409
C00912=1012.630,-115.764,-105.840,165.184,72.239,163.381
C00913=1012.631,-116.014,-105.820,165.166,72.165,163.352
C00914=1012.632,-116.264,-105.802,165.148,72.089,163.324
C00915=1012.634,-116.512,-105.783,165.131,72.013,163.295
C00916=1012.635,-116.762,-105.764,165.113,71.935,163.267
C00917=1012.636,-117.011,-105.744,165.097,71.858,163.239
C00918=1012.638,-117.260,-105.725,165.079,71.780,163.210
C00919=1012.639,-117.509,-105.706,165.063,71.701,163.182
C00920=1012.640,-117.759,-105.687,165.046,71.622,163.153
C00921=1012.641,-118.008,-105.667,165.028,71.542,163.124
C00922=1012.642,-118.257,-105.648,165.011,71.461,163.096
C00923=1012.644,-118.507,-105.630,164.997,71.380,163.068
C00924=1012.645,-118.756,-105.610,164.981,71.298,163.040
C00925=1012.646,-119.005,-105.591,164.964,71.216,163.011
C00926=1012.647,-119.255,-105.572,164.948,71.133,162.983
C00927=1012.648,-119.504,-105.553,164.932,71.049,162.955
C00928=1012.650,-119.753,-105.534,164.917,70.966,162.927
C00929=1012.651,-120.002,-105.515,164.902,70.881,162.898
C00930=1012.652,-120.252,-105.495,164.887,70.795,162.871
C00931=1012.654,-120.500,-105.476,164.872,70.710,162.842
C00932=1012.655,-120.750,-105.457,164.857,70.623,162.814
C00933=1012.657,-120.999,-105.437,164.843,70.536,162.787
C00934=1012.658,-121.248,-105.418,164.828,70.449,162.758
C00935=1012.659,-121.498,-105.399,164.814,70.360,162.730
C00936=1012.661,-121.746,-105.380,164.799,70.273,162.702
C00937=1012.662,-121.996,-105.360,164.786,70.183,162.675
C00938=1012.664,-122.245,-105.341,164.771,70.094,162.647
C00939=1012.665,-122.494,-105.322,164.758,70.003,162.619
C00940=1012.667,-122.744,-105.302,164.746,69.913,162.592
C00941=1012.668,-122.993,-105.283,164.731,69.821,162.564
C00942=1012.669,-123.242,-105.263,164.719,69.730,162.537
C00943=1012.672,-123.491,-105.244,164.708,69.637,162.510
C00944=1012.673,-123.740,-105.225,164.694,69.545,162.482
C00945=1012.674,-123.989,-105.206,164.681,69.451,162.454
C00946=1012.676,-124.239,-105.186,164.670,69.357,162.428
C00947=1012.677,-124.488,-105.166,164.658,69.262,162.400
C00948=1012.680,-124.737,-105.147,164.646,69.167,162.373
C00949=1012.681,-124.987,-105.128,164.635,69.072,162.346
C00950=1012.683,-125.236,-105.108,164.624,68.976,162.320
C00951=1012.684,-125.485,-105.089,164.611,68.879,162.292
C00952=1012.686,-125.734,-105.069,164.602,68.782,162.266
C00953=1012.687,-125.984,-105.050,164.590,68.684,162.238
C00954=1012.690,-126.233,-105.030,164.580,68.586,162.212
C00955=1012.691,-126.482,-105.010,164.570,68.487,162.185
C00956=1012.693,-126.731,-104.991,164.560,68.388,162.159
C00957=1012.695,-126.981,-104.971,164.550,68.288,162.132
C00958=1012.697,-127.230,-104.952,164.540,68.187,162.106
C00959=1012.698,-127.479,-104.932,164.532,68.086,162.080
C00960=1012.700,-127.728,-104.912,164.523,67.984,162.053
C00961=1012.703,-127.977,-104.893,164.514,67.883,162.027
C00962=1012.704,-128.226,-104.873,164.505,67.780,162.001
C00963=1012.706,-128.475,-104.854,164.497,67.676,161.975
C00964=1012.708,-128.725,-104.834,164.489,67.573,161.949
C00965=1012.710,-128.974,-104.814,164.480,67.468,161.922
C00966=1012.712,-129.224,-104.795,164.472,67.363,161.896
C00967=1012.714,-129.472,-104.776,164.464,67.257,161.870
C00968=1012.716,-129.721,-104.756,164.458,67.151,161.845
C00969=1012.718,-129.971,-104.736,164.450,67.044,161.819
C00970=1012.720,-130.220,-104.717,164.443,66.936,161.793
C00971=1012.722,-130.469,-104.697,164.436,66.828,161.767
C00972=1012.724,-130.718,-104.676,164.430,66.720,161.742
C00973=1012.726,-130.967,-104.657,164.423,66.610,161.716
C00974=1012.729,-131.216,-104.637,164.418,66.500,161.690
C00975=1012.730,-131.466,-104.617,164.413,66.390,161.665
C00976=1012.733,-131.715,-104.598,164.406,66.278,161.639
C00977=1012.735,-131.964,-104.578,164.402,66.166,161.614
C00978=1012.737,-132.214,-104.558,164.397,66.054,161.588
C00979=1012.739,-132.463,-104.539,164.392,65.941,161.563
C00980=1012.742,-132.712,-104.519,164.387,65.827,161.538
C00981=1012.744,-132.961,-104.498,164.383,65.712,161.512
C00982=1012.746,-133.210,-104.478,164.378,65.597,161.487
C00983=1012.748,-133.459,-104.459,164.374,65.481,161.461
C00984=1012.753,-133.834,-104.429,164.369,65.306,161.424
C00985=1012.753,-133.960,-104.419,164.367,65.246,161.411
C00986=1012.615,120.124,-124.963,166.115,58.535,160.637
C00987=1012.614,119.896,-124.944,166.105,58.617,160.651
C00988=1012.613,119.668,-124.925,166.096,58.699,160.665
C00989=1012.611,119.432,-124.905,166.087,58.784,160.680
C00990=1012.610,119.198,-124.885,166.077,58.868,160.694
C00991=1012.608,118.963,-124.865,166.067,58.952,160.709
C00992=1012.607,118.728,-124.845,166.057,59.037,160.723
C00993=1012.605,118.492,-124.825,166.047,59.121,160.738
C00994=1012.605,118.257,-124.805,166.038,59.205,160.752
C00995=1012.603,118.021,-124.785,166.029,59.289,160.767
C00996=1012.602,117.787,-124.765,166.020,59.373,160.782
C00997=1012.600,117.551,-124.745,166.011,59.457,160.796
C00998=1012.599,117.316,-124.726,166.002,59.541,160.811
C00999=1012.597,117.081,-124.706,165.994,59.625,160.826
C01000=1012.596,116.846,-124.686,165.985,59.708,160.840
C01001=1012.595,116.611,-124.667,165.977,59.792,160.855
C01002=1012.594,116.375,-124.647,165.968,59.875,160.870
C01003=1012.592,116.141,-124.627,165.959,59.958,160.884
C01004=1012.591,115.905,-124.607,165.952,60.041,160.899
C01005=1012.590,115.670,-124.587,165.943,60.124,160.914
C01006=1012.588,115.435,-124.567,165.935,60.208,160.928
C01007=1012.588,115.199,-124.547,165.926,60.290,160.943
C01008=1012.587,114.965,-124.528,165.919,60.373,160.958
C01009=1012.585,114.729,-124.508,165.910,60.455,160.972
C01010=1012.584,114.494,-124.488,165.903,60.538,160.988
C01011=1012.582,114.259,-124.468,165.895,60.621,161.002
C01012=1012.581,114.024,-124.449,165.888,60.703,161.017
C01013=1012.580,113.789,-124.429,165.880,60.786,161.032
C01014=1012.578,113.553,-124.409,165.873,60.867,161.047
C01015=1012.577,113.318,-124.389,165.864,60.949,161.061
C01016=1012.577,113.083,-124.369,165.858,61.031,161.076
C01017=1012.575,112.848,-124.349,165.851,61.113,161.091
C01018=1012.574,112.613,-124.330,165.844,61.195,161.107
C01019=1012.573,112.378,-124.310,165.836,61.276,161.121
C01020=1012.571,112.142,-124.290,165.830,61.358,161.136
C01021=1012.570,111.908,-124.270,165.823,61.439,161.151
C01022=1012.569,111.673,-124.251,165.817,61.521,161.166
C01023=1012.568,111.437,-124.230,165.810,61.601,161.181
C01024=1012.567,111.202,-124.211,165.804,61.683,161.196
C01025=1012.566,110.967,-124.191,165.798,61.764,161.211
C01026=1012.564,110.732,-124.171,165.791,61.844,161.226
C01027=1012.563,110.497,-124.151,165.785,61.925,161.241
C01028=1012.562,110.261,-124.133,165.779,62.005,161.257
C01029=1012.562,110.026,-124.112,165.773,62.086,161.272
C01030=1012.560,109.791,-124.092,165.767,62.166,161.287
C01031=1012.559,109.556,-124.073,165.762,62.246,161.302
C01032=1012.558,109.321,-124.053,165.755,62.326,161.317
C01033=1012.556,109.085,-124.033,165.751,62.407,161.333
C01034=1012.555,108.851,-124.014,165.745,62.487,161.348
C01035=1012.555,108.615,-123.993,165.739,62.566,161.363
C01036=1012.554,108.380,-123.975,165.734,62.646,161.378
C01037=1012.552,108.144,-123.955,165.729,62.725,161.393
C01038=1012.551,107.909,-123.935,165.724,62.804,161.409
C01039=1012.551,107.674,-123.915,165.719,62.883,161.424
C01040=1012.550,107.439,-123.895,165.714,62.963,161.440
C01041=1012.548,107.204,-123.875,165.709,63.042,161.455
C01042=1012.547,106.969,-123.856,165.705,63.121,161.471
C01043=1012.546,106.734,-123.837,165.700,63.200,161.486
C01044=1012.546,106.498,-123.816,165.695,63.278,161.501
C01045=1012.545,106.264,-123.797,165.692,63.356,161.517
C01046=1012.543,106.028,-123.777,165.687,63.435,161.532
C01047=1012.542,105.793,-123.757,165.682,63.513,161.548
C01048=1012.541,105.558,-123.737,165.679,63.591,161.563
C01049=1012.541,105.323,-123.718,165.675,63.669,161.579
C01050=1012.540,105.088,-123.699,165.671,63.748,161.595
C01051=1012.539,104.852,-123.678,165.668,63.825,161.610
C01052=1012.538,104.617,-123.658,165.664,63.902,161.626
C01053=1012.536,104.255,-123.629,165.658,64.021,161.650
C01054=1012.535,103.911,-123.600,165.654,64.134,161.673
C01055=1012.534,103.676,-123.580,165.651,64.211,161.689
C01056=1012.532,103.441,-123.560,165.648,64.288,161.705
C01057=1012.532,103.205,-123.541,165.645,64.365,161.721
C01058=1012.531,102.970,-123.521,165.641,64.441,161.737
C01059=1012.530,102.736,-123.502,165.639,64.518,161.753
C01060=1012.530,102.500,-123.481,165.636,64.595,161.769
C01061=1012.528,102.264,-123.462,165.634,64.671,161.785
C01062=1012.527,102.029,-123.442,165.631,64.747,161.801
C01063=1012.527,101.794,-123.422,165.628,64.823,161.816
C01064=1012.526,101.559,-123.403,165.627,64.899,161.833
C01065=1012.525,101.324,-123.384,165.624,64.975,161.849
C01066=1012.525,101.089,-123.364,165.622,65.051,161.865
C01067=1012.524,100.854,-123.344,165.620,65.125,161.881
C01068=1012.522,100.618,-123.324,165.619,65.201,161.898
C01069=1012.522,100.383,-123.304,165.617,65.276,161.914
C01070=1012.521,100.148,-123.285,165.615,65.351,161.930
C01071=1012.520,99.912,-123.265,165.614,65.426,161.946
C01072=1012.520,99.677,-123.246,165.613,65.501,161.963
C01073=1012.519,99.442,-123.226,165.611,65.575,161.979
C01074=1012.518,99.207,-123.206,165.610,65.650,161.996
C01075=1012.517,98.972,-123.187,165.610,65.724,162.012
C01076=1012.516,98.736,-123.167,165.607,65.798,162.028
C01077=1012.515,98.501,-123.147,165.606,65.873,162.045
C01078=1012.515,98.265,-123.127,165.607,65.947,162.062
C01079=1012.514,98.030,-123.108,165.606,66.020,162.078
C01080=1012.513,97.795,-123.088,165.605,66.094,162.095
C01081=1012.513,97.560,-123.069,165.604,66.168,162.112
C01082=1012.512,97.325,-123.049,165.604,66.241,162.128
C01083=1012.512,97.090,-123.029,165.604,66.314,162.145
C01084=1012.511,96.854,-123.010,165.604,66.387,162.162
C01085=1012.510,96.618,-122.990,165.603,66.460,162.178
C01086=1012.509,96.383,-122.970,165.604,66.532,162.196
C01087=1012.509,96.148,-122.950,165.605,66.606,162.213
C01088=1012.508,95.913,-122.931,165.604,66.678,162.229
C01089=1012.507,95.678,-122.911,165.606,66.751,162.247
C01090=1012.506,95.442,-122.892,165.606,66.823,162.264
C01091=1012.506,95.207,-122.872,165.607,66.895,162.281
C01092=1012.505,94.971,-122.853,165.607,66.966,162.298
C01093=1012.505,94.736,-122.832,165.609,67.038,162.315
C01094=1012.504,94.501,-122.813,165.610,67.110,162.332
C01095=1012.504,94.266,-122.793,165.611,67.181,162.349
C01096=1012.502,94.030,-122.773,165.612,67.252,162.367
C01097=1012.502,93.794,-122.754,165.614,67.324,162.384
C01098=1012.501,93.559,-122.734,165.614,67.395,162.401
C01099=1012.501,93.324,-122.714,165.616,67.466,162.419
C01100=1012.500,93.089,-122.695,165.618,67.537,162.437
C01101=1012.499,92.854,-122.675,165.620,67.607,162.454
C01102=1012.499,92.618,-122.656,165.622,67.678,162.472
C01103=1012.498,92.383,-122.636,165.624,67.748,162.489
C01104=1012.498,92.147,-122.616,165.627,67.818,162.507
C01105=1012.497,91.912,-122.597,165.628,67.888,162.525
C01106=1012.497,91.677,-122.577,165.630,67.958,162.542
C01107=1012.495,91.441,-122.557,165.633,68.028,162.560
C01108=1012.495,91.206,-122.537,165.636,68.097,162.578
C01109=1012.494,90.946,-122.516,165.639,68.173,162.598
C01110=1012.495,90.627,-122.489,165.642,68.268,162.622
C01111=1012.494,90.293,-122.462,165.646,68.365,162.647
C01112=1012.493,90.010,-122.438,165.651,68.448,162.670
C01113=1012.492,89.772,-122.418,165.654,68.518,162.688
C01114=1012.491,89.540,-122.398,165.658,68.586,162.706
C01115=1012.491,89.311,-122.380,165.662,68.652,162.724
C01116=1012.491,89.083,-122.360,165.665,68.718,162.741
C01117=1012.490,88.859,-122.341,165.669,68.782,162.759
C01118=1012.489,88.635,-122.323,165.672,68.847,162.776
C01119=1012.489,88.411,-122.304,165.676,68.911,162.794
C01120=1012.489,88.186,-122.286,165.680,68.976,162.812
C01121=1012.488,87.959,-122.267,165.683,69.041,162.829
C01122=1012.487,87.728,-122.247,165.688,69.107,162.848
C01123=1012.488,87.495,-122.228,165.693,69.174,162.867
C01124=1012.487,87.259,-122.208,165.699,69.242,162.886
C01125=1012.487,87.020,-122.188,165.702,69.309,162.904
C01126=1012.486,86.781,-122.168,165.707,69.376,162.923
C01127=1012.485,86.542,-122.148,165.712,69.444,162.942
C01128=1012.485,86.172,-122.117,165.720,69.549,162.972
C01129=1012.484,85.822,-122.088,165.728,69.647,163.001
C01130=1012.483,85.582,-122.068,165.735,69.714,163.021
C01131=1012.483,85.341,-122.048,165.739,69.782,163.040
C01132=1012.482,85.099,-122.027,165.745,69.849,163.060
C01133=1012.482,84.857,-122.008,165.752,69.917,163.080
C01134=1012.482,84.615,-121.987,165.758,69.984,163.100
C01135=1012.481,84.371,-121.967,165.765,70.051,163.120
C01136=1012.481,84.128,-121.946,165.771,70.118,163.140
C01137=1012.481,83.884,-121.926,165.777,70.186,163.161
C01138=1012.480,83.639,-121.906,165.783,70.252,163.181
C01139=1012.480,83.394,-121.886,165.790,70.320,163.201
C01140=1012.479,83.148,-121.865,165.798,70.387,163.222
C01141=1012.479,82.903,-121.844,165.804,70.454,163.243
C01142=1012.479,82.657,-121.824,165.813,70.521,163.264
C01143=1012.478,82.411,-121.803,165.820,70.587,163.285
C01144=1012.477,82.164,-121.782,165.827,70.654,163.306
C01145=1012.477,81.917,-121.762,165.835,70.721,163.327
C01146=1012.477,81.670,-121.741,165.843,70.787,163.348
C01147=1012.477,81.426,-121.721,165.851,70.853,163.369
C01148=1012.477,81.199,-121.702,165.858,70.914,163.388
C01149=1012.476,80.981,-121.683,165.866,70.972,163.408
C01150=1012.476,80.764,-121.665,165.873,71.030,163.426
C01151=1012.476,80.535,-121.646,165.880,71.090,163.446
C01152=1012.475,80.292,-121.626,165.889,71.155,163.467
C01153=1012.475,80.046,-121.605,165.899,71.220,163.489
C01154=1012.474,79.801,-121.585,165.906,71.284,163.510
C01155=1012.474,79.559,-121.564,165.916,71.348,163.532
C01156=1012.474,79.319,-121.544,165.924,71.411,163.553
C01157=1012.474,79.082,-121.525,165.933,71.473,163.574
C01158=1012.473,78.847,-121.505,165.943,71.534,163.595
C01159=1012.473,78.614,-121.486,165.951,71.594,163.616
C01160=1012.473,78.384,-121.466,165.961,71.654,163.636
C01161=1012.472,78.155,-121.447,165.970,71.713,163.657
C01162=1012.472,77.928,-121.428,165.979,71.772,163.677
C01163=1012.472,77.701,-121.409,165.987,71.830,163.698
C01164=1012.472,77.473,-121.390,165.997,71.889,163.719
C01165=1012.471,77.244,-121.371,166.006,71.947,163.739
C01166=1012.471,77.014,-121.352,166.017,72.006,163.760
C01167=1012.471,76.781,-121.333,166.027,72.066,163.782
C01168=1012.471,76.545,-121.313,166.038,72.125,163.804
C01169=1012.470,76.307,-121.293,166.048,72.186,163.826
C01170=1012.470,76.066,-121.273,166.058,72.246,163.848
C01171=1012.470,75.823,-121.252,166.069,72.307,163.870
C01172=1012.470,75.577,-121.231,166.080,72.369,163.893
C01173=1012.470,75.329,-121.211,166.092,72.431,163.916
C01174=1012.469,75.080,-121.190,166.103,72.493,163.939
C01175=1012.469,74.821,-121.169,166.116,72.557,163.964
C01176=1012.469,74.548,-121.146,166.129,72.624,163.990
C01177=1012.469,74.282,-121.123,166.142,72.690,164.015
C01178=1012.469,74.030,-121.102,166.154,72.753,164.039
C01179=1012.468,73.784,-121.081,166.167,72.813,164.063
C01180=1012.468,73.538,-121.062,166.178,72.873,164.086
C01181=1012.468,73.293,-121.041,166.193,72.933,164.110
C01182=1012.467,73.049,-121.020,166.204,72.993,164.134
C01183=1012.468,72.805,-121.000,166.216,73.051,164.157
C01184=1012.467,72.563,-120.980,166.231,73.110,164.181
C01185=1012.467,72.320,-120.959,166.244,73.169,164.205
C01186=1012.467,72.078,-120.939,166.255,73.226,164.227
C01187=1012.467,71.837,-120.919,166.269,73.284,164.251
C01188=1012.466,71.595,-120.899,166.283,73.342,164.276
C01189=1012.466,71.354,-120.879,166.296,73.400,164.299
C01190=1012.466,71.113,-120.859,166.309,73.457,164.323
C01191=1012.466,70.872,-120.839,166.324,73.513,164.348
C01192=1012.465,70.631,-120.818,166.336,73.570,164.371
C01193=1012.465,70.390,-120.798,166.350,73.627,164.395
C01194=1012.465,70.149,-120.778,166.364,73.683,164.419
C01195=1012.465,69.908,-120.758,166.380,73.740,164.444
C01196=1012.465,69.666,-120.738,166.394,73.796,164.469
C01197=1012.465,69.423,-120.717,166.407,73.853,164.493
C01198=1012.465,69.177,-120.696,166.424,73.909,164.519
C01199=1012.465,68.929,-120.675,166.438,73.966,164.543
C01200=1012.465,68.679,-120.655,166.454,74.024,164.569
C01201=1012.464,68.431,-120.634,166.470,74.081,164.595
C01202=1012.464,68.185,-120.613,166.486,74.137,164.621
C01203=1012.464,67.944,-120.593,166.500,74.193,164.645
C01204=1012.464,67.704,-120.573,166.515,74.246,164.670
C01205=1012.464,67.467,-120.554,166.530,74.300,164.695
C01206=1012.464,67.230,-120.533,166.546,74.354,164.720
C01207=1012.464,66.993,-120.514,166.562,74.407,164.745
C01208=1012.464,66.757,-120.494,166.577,74.460,164.769
C01209=1012.464,66.543,-120.476,166.592,74.508,164.792
C01210=1012.464,66.152,-120.443,166.617,74.594,164.833
C01211=1012.463,65.919,-120.423,166.634,74.647,164.859
C01212=1012.464,65.676,-120.403,166.652,74.700,164.885
C01213=1012.463,65.423,-120.382,166.669,74.756,164.912
C01214=1012.463,65.162,-120.361,166.687,74.813,164.940
C01215=1012.463,64.897,-120.338,166.706,74.871,164.969
C01216=1012.463,64.626,-120.316,166.725,74.930,164.998
C01217=1012.463,64.360,-120.293,166.746,74.987,165.028
C01218=1012.463,63.974,-120.261,166.772,75.071,165.070
C01219=1012.463,63.618,-120.231,166.799,75.148,165.110
C01220=1012.463,63.335,-120.207,166.821,75.208,165.141
C01221=1012.463,63.039,-120.183,166.842,75.271,165.173
C01222=1012.463,62.764,-120.159,166.863,75.330,165.204
C01223=1012.462,62.476,-120.135,166.886,75.390,165.236
C01224=1012.463,62.200,-120.112,166.908,75.448,165.268
C01225=1012.462,61.964,-120.093,166.924,75.498,165.294
C01226=1012.462,61.728,-120.073,166.943,75.547,165.320
C01227=1012.462,61.493,-120.053,166.963,75.596,165.348
C01228=1012.462,61.257,-120.033,166.982,75.645,165.375
C01229=1012.463,61.021,-120.013,166.999,75.693,165.401
C01230=1012.463,60.785,-119.994,167.018,75.742,165.428
C01231=1012.463,60.549,-119.974,167.039,75.790,165.456
C01232=1012.462,60.314,-119.954,167.057,75.839,165.483
C01233=1012.462,60.078,-119.935,167.078,75.887,165.511
C01234=1012.462,59.842,-119.915,167.097,75.935,165.538
C01235=1012.462,59.606,-119.895,167.117,75.983,165.566
C01236=1012.462,59.370,-119.875,167.137,76.030,165.594
C01237=1012.462,59.135,-119.855,167.155,76.077,165.620
C01238=1012.462,58.899,-119.836,167.176,76.125,165.648
C01239=1012.462,58.663,-119.816,167.197,76.173,165.677
C01240=1012.462,58.427,-119.796,167.217,76.219,165.705
C01241=1012.462,58.191,-119.777,167.237,76.266,165.732
C01242=1012.462,57.956,-119.756,167.258,76.312,165.760
C01243=1012.462,57.720,-119.737,167.279,76.358,165.789
C01244=1012.462,57.485,-119.717,167.299,76.405,165.817
C01245=1012.463,57.248,-119.697,167.321,76.451,165.846
C01246=1012.463,57.013,-119.678,167.340,76.497,165.873
C01247=1012.462,56.777,-119.658,167.364,76.543,165.903
C01248=1012.462,56.542,-119.638,167.384,76.588,165.931
C01249=1012.462,56.306,-119.619,167.406,76.633,165.960
C01250=1012.463,56.070,-119.599,167.427,76.679,165.989
C01251=1012.463,55.834,-119.579,167.450,76.724,166.018
C01252=1012.462,55.599,-119.559,167.472,76.769,166.048
C01253=1012.462,55.363,-119.539,167.493,76.813,166.076
C01254=1012.462,55.127,-119.520,167.517,76.858,166.106
C01255=1012.463,54.891,-119.500,167.538,76.902,166.135
C01256=1012.463,54.655,-119.480,167.562,76.947,166.165
C01257=1012.462,54.420,-119.460,167.584,76.992,166.194
C01258=1012.462,54.184,-119.441,167.607,77.035,166.224
C01259=1012.463,53.948,-119.421,167.628,77.078,166.253
C01260=1012.463,53.713,-119.401,167.651,77.122,166.282
C01261=1012.463,53.477,-119.382,167.675,77.166,166.313
C01262=1012.463,53.242,-119.361,167.698,77.209,166.342
C01263=1012.463,53.006,-119.342,167.720,77.252,166.372
C01264=1012.463,52.770,-119.322,167.746,77.295,166.404
C01265=1012.463,52.534,-119.302,167.769,77.338,166.434
C01266=1012.463,52.299,-119.282,167.793,77.381,166.464
C01267=1012.463,52.063,-119.263,167.815,77.422,166.493
C01268=1012.464,51.827,-119.243,167.840,77.464,166.524
C01269=1012.463,51.591,-119.223,167.866,77.507,166.556
C01270=1012.463,51.355,-119.204,167.889,77.548,166.585
C01271=1012.463,51.120,-119.183,167.913,77.590,166.616
C01272=1012.463,50.884,-119.164,167.937,77.631,166.646
C01273=1012.464,50.648,-119.144,167.961,77.673,166.677
C01274=1012.464,50.412,-119.124,167.987,77.714,166.708
C01275=1012.463,50.177,-119.104,168.011,77.756,166.739
C01276=1012.463,49.941,-119.085,168.037,77.797,166.771
C01277=1012.463,49.706,-119.065,168.062,77.837,166.802
C01278=1012.464,49.470,-119.045,168.088,77.878,166.834
C01279=1012.463,49.234,-119.025,168.113,77.918,166.865
C01280=1012.464,48.999,-119.006,168.138,77.958,166.896
C01281=1012.464,48.763,-118.986,168.163,77.998,166.928
C01282=1012.465,48.527,-118.966,168.190,78.038,166.960
C01283=1012.464,48.292,-118.946,168.216,78.078,166.992
C01284=1012.464,48.056,-118.927,168.240,78.117,167.022
C01285=1012.464,47.821,-118.907,168.268,78.157,167.055
C01286=1012.464,47.585,-118.887,168.292,78.196,167.086
C01287=1012.465,47.349,-118.867,168.318,78.235,167.117
C01288=1012.464,47.114,-118.847,168.347,78.274,167.152
C01289=1012.465,46.878,-118.828,168.373,78.313,167.184
C01290=1012.465,46.643,-118.808,168.397,78.351,167.214
C01291=1012.465,46.407,-118.788,168.425,78.389,167.247
C01292=1012.465,46.171,-118.769,168.452,78.428,167.280
C01293=1012.465,45.936,-118.749,168.478,78.465,167.312
C01294=1012.465,45.700,-118.729,168.507,78.504,167.346
C01295=1012.465,45.465,-118.709,168.534,78.541,167.378
C01296=1012.466,45.229,-118.690,168.560,78.579,167.410
C01297=1012.466,44.994,-118.669,168.587,78.616,167.443
C01298=1012.466,44.758,-118.650,168.616,78.653,167.476
C01299=1012.466,44.523,-118.630,168.644,78.690,167.509
C01300=1012.465,44.287,-118.610,168.670,78.726,167.541
C01301=1012.466,44.051,-118.590,168.698,78.764,167.575
C01302=1012.467,43.816,-118.571,168.725,78.800,167.607
C01303=1012.466,43.581,-118.551,168.755,78.837,167.642
C01304=1012.466,43.345,-118.531,168.783,78.873,167.675
C01305=1012.466,43.109,-118.512,168.812,78.908,167.709
C01306=1012.466,42.874,-118.491,168.840,78.945,167.742
C01307=1012.467,42.639,-118.472,168.866,78.980,167.773
C01308=1012.467,42.403,-118.453,168.896,79.015,167.808
C01309=1012.467,42.168,-118.432,168.926,79.051,167.843
C01310=1012.467,41.932,-118.413,168.952,79.086,167.875
C01311=1012.467,41.696,-118.393,168.980,79.121,167.908
C01312=1012.467,41.462,-118.373,169.011,79.156,167.944
C01313=1012.467,41.226,-118.353,169.041,79.190,167.978
C01314=1012.467,40.990,-118.334,169.070,79.225,168.012
C01315=1012.467,40.755,-118.314,169.096,79.259,168.043
C01316=1012.468,40.519,-118.294,169.127,79.293,168.078
C01317=1012.468,40.284,-118.275,169.158,79.327,168.114
C01318=1012.468,40.048,-118.254,169.185,79.361,168.146
C01319=1012.468,39.813,-118.235,169.216,79.395,168.182
C01320=1012.468,39.577,-118.215,169.245,79.428,168.215
C01321=1012.469,39.342,-118.195,169.276,79.461,168.250
C01322=1012.469,39.106,-118.175,169.305,79.494,168.284
C01323=1012.469,38.871,-118.156,169.335,79.528,168.319
C01324=1012.469,38.636,-118.136,169.366,79.560,168.354
C01325=1012.469,38.400,-118.117,169.395,79.592,168.387
C01326=1012.469,38.165,-118.096,169.425,79.626,168.422
C01327=1012.469,37.929,-118.076,169.454,79.658,168.456
C01328=1012.470,37.694,-118.057,169.483,79.690,168.490
C01329=1012.469,37.459,-118.037,169.513,79.721,168.524
C01330=1012.469,37.223,-118.018,169.544,79.753,168.559
C01331=1012.470,36.987,-117.998,169.574,79.785,168.594
C01332=1012.470,36.752,-117.978,169.606,79.816,168.629
C01333=1012.470,36.517,-117.958,169.637,79.848,168.664
C01334=1012.470,36.281,-117.938,169.666,79.878,168.698
C01335=1012.470,36.046,-117.919,169.698,79.910,168.734
C01336=1012.471,35.810,-117.899,169.728,79.940,168.768
C01337=1012.471,35.575,-117.879,169.758,79.971,168.802
C01338=1012.471,35.340,-117.860,169.788,80.001,168.837
C01339=1012.471,35.105,-117.839,169.820,80.031,168.872
C01340=1012.471,34.869,-117.820,169.850,80.061,168.907
C01341=1012.472,34.634,-117.800,169.883,80.091,168.943
C01342=1012.472,34.399,-117.780,169.915,80.121,168.979
C01343=1012.472,34.163,-117.760,169.945,80.150,169.013
C01344=1012.471,33.928,-117.740,169.975,80.179,169.047
C01345=1012.472,33.693,-117.721,170.008,80.209,169.084
C01346=1012.472,33.457,-117.702,170.038,80.238,169.118
C01347=1012.472,33.221,-117.681,170.070,80.267,169.154
C01348=1012.473,32.986,-117.662,170.101,80.296,169.189
C01349=1012.472,32.751,-117.642,170.134,80.324,169.225
C01350=1012.472,32.515,-117.622,170.162,80.353,169.257
C01351=1012.473,32.280,-117.603,170.195,80.381,169.294
C01352=1012.473,32.045,-117.582,170.224,80.409,169.327
C01353=1012.474,31.810,-117.563,170.259,80.436,169.365
C01354=1012.473,31.574,-117.543,170.290,80.464,169.399
C01355=1012.473,31.339,-117.523,170.320,80.492,169.434
C01356=1012.474,31.104,-117.504,170.352,80.519,169.469
C01357=1012.474,30.868,-117.484,170.384,80.546,169.504
C01358=1012.474,30.632,-117.464,170.416,80.573,169.540
C01359=1012.474,30.317,-117.438,170.456,80.609,169.585
C01360=1012.474,29.927,-117.404,170.509,80.653,169.643
C01361=1012.475,29.692,-117.385,170.540,80.679,169.678
C01362=1012.475,29.456,-117.365,170.571,80.705,169.712
C01363=1012.475,29.221,-117.345,170.605,80.732,169.749
C01364=1012.476,28.985,-117.326,170.634,80.757,169.782
C01365=1012.476,28.751,-117.306,170.666,80.782,169.817
C01366=1012.475,28.516,-117.286,170.699,80.808,169.853
C01367=1012.476,28.282,-117.266,170.728,80.833,169.886
C01368=1012.476,28.048,-117.247,170.762,80.858,169.922
C01369=1012.476,27.813,-117.227,170.793,80.882,169.956
C01370=1012.477,27.580,-117.207,170.823,80.907,169.990
C01371=1012.476,27.346,-117.188,170.855,80.932,170.025
C01372=1012.476,27.112,-117.168,170.886,80.956,170.059
C01373=1012.477,26.877,-117.149,170.917,80.981,170.094
C01374=1012.476,26.642,-117.129,170.949,81.005,170.129
C01375=1012.477,26.405,-117.109,170.982,81.029,170.164
C01376=1012.478,26.168,-117.089,171.011,81.052,170.197
C01377=1012.478,25.931,-117.069,171.045,81.076,170.233
C01378=1012.477,25.694,-117.049,171.075,81.099,170.266
C01379=1012.477,25.457,-117.029,171.108,81.123,170.302
C01380=1012.478,25.222,-117.010,171.140,81.146,170.337
C01381=1012.478,24.986,-116.990,171.171,81.169,170.371
C01382=1012.479,24.750,-116.970,171.203,81.192,170.405
C01383=1012.478,24.515,-116.950,171.231,81.214,170.437
C01384=1012.479,24.283,-116.931,171.263,81.236,170.472
C01385=1012.479,24.061,-116.912,171.289,81.257,170.501
C01386=1012.479,23.852,-116.895,171.319,81.276,170.532
C01387=1012.479,23.487,-116.864,171.365,81.310,170.583
C01388=1012.479,23.186,-116.838,171.405,81.337,170.626
C01389=1012.480,22.895,-116.814,171.446,81.364,170.670
C01390=1012.480,22.550,-116.785,171.489,81.395,170.717
C01391=1012.480,22.137,-116.750,171.543,81.432,170.775
C01392=1012.480,21.726,-116.715,171.594,81.467,170.831
C01393=1012.481,21.466,-116.694,171.629,81.490,170.868
C01394=1012.481,21.177,-116.670,171.664,81.515,170.908
C01395=1012.481,20.868,-116.644,171.704,81.540,170.950
C01396=1012.482,20.549,-116.617,171.743,81.567,170.993
C01397=1012.482,20.229,-116.590,171.786,81.594,171.039
C01398=1012.482,19.929,-116.565,171.825,81.618,171.080
C01399=1012.482,19.533,-116.532,171.871,81.649,171.130
C01400=1012.483,19.228,-116.506,171.908,81.674,171.171
C01401=1012.483,18.967,-116.485,171.940,81.694,171.205
C01402=1012.483,18.733,-116.464,171.968,81.712,171.236
C01403=1012.483,18.499,-116.445,171.999,81.730,171.268
C01404=1012.483,18.266,-116.425,172.029,81.748,171.300
C01405=1012.484,18.034,-116.406,172.055,81.765,171.328
C01406=1012.484,17.803,-116.386,172.081,81.782,171.357
C01407=1012.484,17.571,-116.367,172.108,81.799,171.386
C01408=1012.484,17.341,-116.347,172.137,81.816,171.416
C01409=1012.484,17.111,-116.328,172.164,81.833,171.446
C01410=1012.485,16.882,-116.309,172.192,81.849,171.476
C01411=1012.485,16.653,-116.290,172.220,81.866,171.505
C01412=1012.485,16.426,-116.271,172.245,81.882,171.532
C01413=1012.485,16.198,-116.251,172.270,81.897,171.559
C01414=1012.485,15.971,-116.232,172.296,81.912,171.587
C01415=1012.485,15.744,-116.213,172.325,81.929,171.618
C01416=1012.485,15.518,-116.194,172.348,81.943,171.643
C01417=1012.486,15.292,-116.176,172.373,81.958,171.670
C01418=1012.486,15.066,-116.157,172.400,81.973,171.699
C01419=1012.486,14.840,-116.137,172.427,81.988,171.727
C01420=1012.486,14.613,-116.119,172.450,82.002,171.752
C01421=1012.486,14.387,-116.099,172.477,82.017,171.780
C01422=1012.487,14.160,-116.080,172.500,82.031,171.806
C01423=1012.486,13.933,-116.061,172.525,82.045,171.832
C01424=1012.487,13.705,-116.042,172.548,82.059,171.857
C01425=1012.487,13.478,-116.023,172.573,82.073,171.883
C01426=1012.487,13.249,-116.004,172.596,82.087,171.908
C01427=1012.487,13.022,-115.985,172.621,82.100,171.935
C01428=1012.488,12.793,-115.966,172.642,82.113,171.957
C01429=1012.488,12.564,-115.946,172.667,82.126,171.984
C01430=1012.488,12.336,-115.927,172.693,82.140,172.010
C01431=1012.488,12.108,-115.908,172.714,82.153,172.033
C01432=1012.488,11.886,-115.889,172.736,82.165,172.057
C01433=1012.489,11.666,-115.871,172.759,82.177,172.081
C01434=1012.489,11.450,-115.852,172.781,82.189,172.105
C01435=1012.489,11.234,-115.834,172.800,82.200,172.125
C01436=1012.489,11.016,-115.816,172.824,82.211,172.150
C01437=1012.490,10.795,-115.798,172.842,82.223,172.170
C01438=1012.489,10.571,-115.778,172.865,82.235,172.194
C01439=1012.489,10.346,-115.760,172.885,82.245,172.215
C01440=1012.490,10.121,-115.741,172.904,82.257,172.236
C01441=1012.491,9.897,-115.722,172.928,82.268,172.261
C01442=1012.490,9.674,-115.703,172.948,82.279,172.282
C01443=1012.491,9.451,-115.685,172.969,82.289,172.304
C01444=1012.490,9.229,-115.666,172.984,82.299,172.321
C01445=1012.491,9.007,-115.647,173.005,82.310,172.343
C01446=1012.491,8.785,-115.629,173.025,82.321,172.364
C01447=1012.491,8.561,-115.610,173.043,82.330,172.383
C01448=1012.492,8.339,-115.591,173.063,82.340,172.404
C01449=1012.491,8.115,-115.573,173.081,82.350,172.423
C01450=1012.492,7.890,-115.553,173.098,82.359,172.442
C01451=1012.491,7.665,-115.534,173.114,82.369,172.460
C01452=1012.492,7.439,-115.516,173.132,82.378,172.478
C01453=1012.492,7.211,-115.496,173.150,82.387,172.497
C01454=1012.492,6.982,-115.477,173.169,82.396,172.516
C01455=1012.492,6.751,-115.458,173.186,82.405,172.535
C01456=1012.493,6.518,-115.439,173.204,82.414,172.554
C01457=1012.493,6.285,-115.419,173.222,82.423,172.573
C01458=1012.493,6.051,-115.399,173.237,82.431,172.589
C01459=1012.493,5.816,-115.379,173.255,82.440,172.608
C01460=1012.493,5.583,-115.359,173.270,82.448,172.624
C01461=1012.494,5.351,-115.340,173.284,82.456,172.640
C01462=1012.494,5.119,-115.321,173.299,82.464,172.655
C01463=1012.494,4.888,-115.301,173.315,82.471,172.672
C01464=1012.494,4.656,-115.282,173.330,82.479,172.688
C01465=1012.495,4.423,-115.262,173.345,82.486,172.704
C01466=1012.495,4.191,-115.243,173.357,82.493,172.716
C01467=1012.495,3.962,-115.224,173.373,82.500,172.733
C01468=1012.495,3.743,-115.205,173.385,82.506,172.746
C01469=1012.495,3.535,-115.188,173.398,82.512,172.759
C01470=1012.495,3.144,-115.155,173.419,82.523,172.781
C01471=1012.496,2.760,-115.123,173.437,82.532,172.801
C01472=1012.496,2.351,-115.088,173.459,82.543,172.824
C01473=1012.497,2.130,-115.070,173.468,82.548,172.833
C01474=1012.497,1.901,-115.051,173.481,82.554,172.847
C01475=1012.497,1.666,-115.031,173.490,82.559,172.857
C01476=1012.497,1.430,-115.011,173.500,82.563,172.867
C01477=1012.497,1.193,-114.991,173.508,82.568,172.876
C01478=1012.497,0.957,-114.971,173.517,82.573,172.886
C01479=1012.498,0.722,-114.951,173.527,82.577,172.896
C01480=1012.497,0.488,-114.932,173.537,82.581,172.906
C01481=1012.498,0.253,-114.912,173.547,82.585,172.917
C01482=1012.498,0.017,-114.892,173.553,82.589,172.923
C01483=1012.498,-0.220,-114.872,173.563,82.593,172.933
C01484=1012.498,-0.458,-114.852,173.568,82.597,172.939
C01485=1012.498,-0.697,-114.832,173.573,82.600,172.945
C01486=1012.499,-0.936,-114.812,173.580,82.603,172.952
C01487=1012.499,-1.176,-114.792,173.587,82.606,172.959
C01488=1012.499,-1.416,-114.771,173.592,82.609,172.965
C01489=1012.499,-1.657,-114.751,173.599,82.612,172.972
C01490=1012.500,-1.899,-114.731,173.607,82.614,172.980
C01491=1012.500,-2.143,-114.711,173.609,82.617,172.983
C01492=1012.500,-2.386,-114.691,173.611,82.619,172.985
C01493=1012.500,-2.629,-114.670,173.619,82.621,172.993
C01494=1012.500,-2.874,-114.649,173.621,82.623,172.996
C01495=1012.500,-3.120,-114.628,173.625,82.624,172.999
C01496=1012.501,-3.362,-114.608,173.624,82.625,172.999
C01497=1012.500,-3.599,-114.588,173.628,82.626,173.003
C01498=1012.501,-3.830,-114.569,173.632,82.627,173.006
C01499=1012.501,-4.056,-114.550,173.630,82.628,173.006
C01500=1012.501,-4.281,-114.531,173.630,82.628,173.006
C01501=1012.501,-4.510,-114.512,173.630,82.628,173.006
C01502=1012.502,-4.745,-114.492,173.635,82.629,173.010
C01503=1012.503,-4.989,-114.472,173.630,82.628,173.006
C01504=1012.502,-5.242,-114.450,173.630,82.628,173.006
C01505=1012.502,-5.498,-114.429,173.630,82.628,173.006
C01506=1012.503,-5.757,-114.407,173.627,82.626,173.002
C01507=1012.503,-6.015,-114.386,173.628,82.626,173.003
C01508=1012.503,-6.273,-114.363,173.625,82.624,172.999
C01509=1012.503,-6.530,-114.342,173.621,82.623,172.996
C01510=1012.503,-6.787,-114.320,173.618,82.622,172.992
C01511=1012.503,-7.044,-114.299,173.610,82.619,172.985
C01512=1012.504,-7.299,-114.278,173.608,82.617,172.982
C01513=1012.504,-7.553,-114.256,173.606,82.615,172.979
C01514=1012.505,-7.807,-114.235,173.598,82.613,172.972
C01515=1012.505,-8.059,-114.214,173.592,82.609,172.965
C01516=1012.505,-8.311,-114.192,173.586,82.607,172.959
C01517=1012.505,-8.563,-114.171,173.579,82.604,172.952
C01518=1012.505,-8.815,-114.150,173.573,82.600,172.945
C01519=1012.505,-9.065,-114.129,173.562,82.597,172.935
C01520=1012.505,-9.317,-114.108,173.557,82.593,172.928
C01521=1012.506,-9.568,-114.086,173.547,82.589,172.918
C01522=1012.506,-9.819,-114.066,173.538,82.584,172.908
C01523=1012.506,-10.069,-114.044,173.528,82.580,172.898
C01524=1012.506,-10.319,-114.024,173.518,82.576,172.888
C01525=1012.507,-10.569,-114.003,173.509,82.571,172.878
C01526=1012.507,-10.819,-113.982,173.500,82.566,172.869
C01527=1012.507,-11.068,-113.961,173.487,82.560,172.855
C01528=1012.507,-11.317,-113.940,173.474,82.554,172.842
C01529=1012.507,-11.565,-113.919,173.465,82.549,172.832
C01530=1012.508,-11.812,-113.898,173.453,82.543,172.819
C01531=1012.508,-12.059,-113.878,173.441,82.537,172.806
C01532=1012.508,-12.305,-113.857,173.423,82.530,172.789
C01533=1012.508,-12.551,-113.836,173.411,82.524,172.776
C01534=1012.508,-12.796,-113.816,173.400,82.517,172.763
C01535=1012.509,-13.037,-113.796,173.383,82.510,172.747
C01536=1012.509,-13.275,-113.775,173.373,82.503,172.735
C01537=1012.509,-13.507,-113.756,173.356,82.496,172.718
C01538=1012.509,-13.737,-113.737,173.340,82.489,172.701
C01539=1012.510,-13.962,-113.717,173.330,82.482,172.689
C01540=1012.510,-14.186,-113.699,173.313,82.475,172.673
C01541=1012.509,-14.410,-113.680,173.298,82.467,172.657
C01542=1012.510,-14.632,-113.661,173.282,82.460,172.640
C01543=1012.510,-14.857,-113.642,173.267,82.452,172.624
C01544=1012.511,-15.084,-113.624,173.248,82.444,172.605
C01545=1012.510,-15.314,-113.604,173.235,82.435,172.590
C01546=1012.510,-15.547,-113.584,173.215,82.427,172.570
C01547=1012.511,-15.782,-113.565,173.198,82.418,172.551
C01548=1012.511,-16.019,-113.545,173.180,82.408,172.532
C01549=1012.511,-16.254,-113.526,173.157,82.399,172.509
C01550=1012.511,-16.489,-113.505,173.140,82.389,172.491
C01551=1012.512,-16.726,-113.486,173.123,82.379,172.472
C01552=1012.512,-16.964,-113.466,173.101,82.370,172.450
C01553=1012.512,-17.198,-113.446,173.081,82.359,172.428
C01554=1012.512,-17.428,-113.426,173.060,82.348,172.406
C01555=1012.513,-17.659,-113.408,173.039,82.338,172.385
C01556=1012.513,-17.907,-113.386,173.019,82.327,172.363
C01557=1012.513,-18.192,-113.363,172.992,82.314,172.335
C01558=1012.514,-18.509,-113.335,172.964,82.298,172.305
C01559=1012.514,-18.841,-113.308,172.931,82.282,172.271
C01560=1012.513,-19.167,-113.280,172.899,82.265,172.237
C01561=1012.514,-19.466,-113.255,172.871,82.250,172.207
C01562=1012.515,-19.727,-113.233,172.845,82.236,172.180
C01563=1012.515,-20.077,-113.204,172.811,82.218,172.144
C01564=1012.515,-20.354,-113.180,172.780,82.202,172.110
C01565=1012.515,-20.588,-113.161,172.757,82.190,172.087
C01566=1012.515,-20.823,-113.141,172.731,82.176,172.060
C01567=1012.516,-21.057,-113.122,172.706,82.163,172.033
C01568=1012.516,-21.291,-113.102,172.682,82.148,172.007
C01569=1012.516,-21.525,-113.082,172.657,82.135,171.980
C01570=1012.516,-21.760,-113.063,172.629,82.120,171.951
C01571=1012.517,-21.993,-113.043,172.603,82.107,171.924
C01572=1012.517,-22.228,-113.023,172.576,82.092,171.895
C01573=1012.517,-22.462,-113.003,172.548,82.077,171.866
C01574=1012.518,-22.695,-112.983,172.526,82.062,171.841
C01575=1012.517,-22.929,-112.964,172.494,82.046,171.809
C01576=1012.517,-23.164,-112.944,172.467,82.031,171.780
C01577=1012.518,-23.398,-112.924,172.441,82.016,171.752
C01578=1012.518,-23.632,-112.905,172.415,82.000,171.724
C01579=1012.518,-23.866,-112.886,172.385,81.984,171.693
C01580=1012.518,-24.101,-112.866,172.355,81.968,171.661
C01581=1012.518,-24.335,-112.846,172.326,81.951,171.630
C01582=1012.519,-24.569,-112.827,172.296,81.935,171.599
C01583=1012.520,-24.803,-112.807,172.268,81.918,171.569
C01584=1012.519,-25.037,-112.787,172.241,81.901,171.539
C01585=1012.519,-25.271,-112.767,172.209,81.883,171.506
C01586=1012.520,-25.505,-112.748,172.181,81.866,171.476
C01587=1012.520,-25.739,-112.728,172.150,81.848,171.443
C01588=1012.520,-25.974,-112.708,172.119,81.831,171.410
C01589=1012.520,-26.208,-112.688,172.089,81.812,171.378
C01590=1012.521,-26.442,-112.669,172.058,81.794,171.345
C01591=1012.521,-26.676,-112.649,172.028,81.776,171.314
C01592=1012.521,-26.911,-112.629,171.995,81.757,171.279
C01593=1012.521,-27.145,-112.610,171.966,81.738,171.247
C01594=1012.522,-27.379,-112.590,171.933,81.719,171.213
C01595=1012.522,-27.613,-112.570,171.902,81.699,171.179
C01596=1012.522,-27.848,-112.551,171.870,81.679,171.145
C01597=1012.522,-28.082,-112.531,171.838,81.660,171.111
C01598=1012.522,-28.316,-112.511,171.803,81.640,171.074
C01599=1012.523,-28.550,-112.492,171.772,81.620,171.041
C01600=1012.523,-28.784,-112.471,171.738,81.599,171.005
C01601=1012.523,-29.018,-112.452,171.705,81.578,170.969
C01602=1012.523,-29.253,-112.432,171.675,81.558,170.937
C01603=1012.523,-29.487,-112.413,171.642,81.537,170.902
C01604=1012.524,-29.721,-112.393,171.606,81.515,170.864
C01605=1012.524,-29.955,-112.373,171.574,81.493,170.829
C01606=1012.524,-30.190,-112.353,171.538,81.471,170.791
C01607=1012.525,-30.424,-112.334,171.507,81.450,170.757
C01608=1012.525,-30.659,-112.314,171.473,81.427,170.721
C01609=1012.526,-30.892,-112.294,171.438,81.405,170.683
C01610=1012.525,-31.126,-112.275,171.404,81.382,170.647
C01611=1012.525,-31.361,-112.255,171.371,81.360,170.611
C01612=1012.526,-31.595,-112.235,171.334,81.336,170.572
C01613=1012.526,-31.830,-112.216,171.302,81.313,170.538
C01614=1012.527,-32.064,-112.196,171.266,81.289,170.499
C01615=1012.527,-32.298,-112.176,171.231,81.265,170.462
C01616=1012.527,-32.532,-112.156,171.195,81.242,170.424
C01617=1012.528,-32.767,-112.137,171.161,81.218,170.387
C01618=1012.527,-33.001,-112.117,171.127,81.193,170.350
C01619=1012.527,-33.235,-112.098,171.091,81.168,170.311
C01620=1012.528,-33.469,-112.078,171.057,81.144,170.274
C01621=1012.529,-33.827,-112.048,171.001,81.105,170.215
C01622=1012.529,-34.173,-112.019,170.950,81.068,170.159
C01623=1012.529,-34.407,-111.999,170.915,81.042,170.121
C01624=1012.530,-34.641,-111.979,170.877,81.016,170.080
C01625=1012.530,-34.875,-111.959,170.844,80.989,170.044
C01626=1012.530,-35.109,-111.940,170.806,80.963,170.004
C01627=1012.530,-35.344,-111.920,170.770,80.936,169.964
C01628=1012.530,-35.578,-111.901,170.734,80.909,169.926
C01629=1012.531,-35.812,-111.881,170.699,80.882,169.887
C01630=1012.531,-36.046,-111.861,170.663,80.855,169.849
C01631=1012.531,-36.281,-111.841,170.625,80.827,169.808
C01632=1012.532,-36.515,-111.822,170.591,80.800,169.770
C01633=1012.533,-36.749,-111.802,170.554,80.772,169.730
C01634=1012.533,-36.984,-111.782,170.517,80.743,169.691
C01635=1012.533,-37.218,-111.762,170.481,80.715,169.651
C01636=1012.532,-37.452,-111.743,170.446,80.686,169.612
C01637=1012.533,-37.686,-111.724,170.407,80.657,169.571
C01638=1012.533,-37.920,-111.703,170.373,80.628,169.533
C01639=1012.534,-38.154,-111.683,170.336,80.598,169.493
C01640=1012.534,-38.389,-111.664,170.298,80.569,169.452
C01641=1012.535,-38.622,-111.644,170.262,80.539,169.413
C01642=1012.535,-38.857,-111.624,170.226,80.509,169.373
C01643=1012.535,-39.091,-111.604,170.188,80.478,169.332
C01644=1012.535,-39.326,-111.585,170.153,80.448,169.293
C01645=1012.535,-39.559,-111.566,170.116,80.417,169.253
C01646=1012.536,-39.794,-111.546,170.078,80.386,169.212
C01647=1012.536,-40.028,-111.526,170.041,80.355,169.172
C01648=1012.537,-40.262,-111.507,170.005,80.324,169.132
C01649=1012.537,-40.496,-111.487,169.968,80.291,169.091
C01650=1012.537,-40.731,-111.467,169.932,80.260,169.051
C01651=1012.538,-40.964,-111.447,169.895,80.227,169.011
C01652=1012.538,-41.198,-111.427,169.857,80.195,168.970
C01653=1012.538,-41.433,-111.407,169.821,80.162,168.929
C01654=1012.538,-41.666,-111.388,169.785,80.130,168.890
C01655=1012.539,-41.901,-111.368,169.750,80.096,168.851
C01656=1012.539,-42.135,-111.349,169.712,80.063,168.809
C01657=1012.540,-42.369,-111.329,169.675,80.029,168.768
C01658=1012.540,-42.603,-111.309,169.640,79.996,168.729
C01659=1012.540,-42.838,-111.289,169.604,79.962,168.689
C01660=1012.541,-43.071,-111.269,169.565,79.927,168.647
C01661=1012.541,-43.305,-111.249,169.531,79.892,168.608
C01662=1012.541,-43.539,-111.230,169.492,79.857,168.566
C01663=1012.541,-43.773,-111.211,169.459,79.823,168.528
C01664=1012.542,-44.007,-111.191,169.421,79.788,168.487
C01665=1012.542,-44.241,-111.171,169.385,79.752,168.447
C01666=1012.542,-44.475,-111.151,169.347,79.716,168.404
C01667=1012.543,-44.709,-111.131,169.311,79.680,168.365
C01668=1012.543,-44.943,-111.112,169.275,79.644,168.324
C01669=1012.543,-45.177,-111.093,169.240,79.608,168.285
C01670=1012.544,-45.411,-111.073,169.204,79.571,168.245
C01671=1012.544,-45.644,-111.053,169.169,79.534,168.205
C01672=1012.544,-45.879,-111.033,169.131,79.496,168.163
C01673=1012.545,-46.112,-111.013,169.096,79.460,168.124
C01674=1012.545,-46.347,-110.994,169.060,79.421,168.083
C01675=1012.546,-46.581,-110.974,169.026,79.384,168.045
C01676=1012.546,-46.813,-110.954,168.991,79.346,168.005
C01677=1012.546,-47.048,-110.935,168.953,79.307,167.963
C01678=1012.547,-47.282,-110.915,168.918,79.268,167.924
C01679=1012.547,-47.516,-110.895,168.884,79.230,167.885
C01680=1012.548,-47.749,-110.875,168.849,79.190,167.845
C01681=1012.548,-47.984,-110.855,168.812,79.151,167.804
C01682=1012.549,-48.217,-110.836,168.777,79.112,167.765
C01683=1012.549,-48.450,-110.816,168.743,79.072,167.725
C01684=1012.549,-48.685,-110.796,168.706,79.031,167.684
C01685=1012.550,-48.918,-110.777,168.673,78.992,167.646
C01686=1012.550,-49.153,-110.757,168.638,78.950,167.606
C01687=1012.551,-49.386,-110.737,168.603,78.910,167.566
C01688=1012.552,-49.620,-110.717,168.569,78.869,167.527
C01689=1012.552,-49.854,-110.698,168.533,78.827,167.486
C01690=1012.552,-50.087,-110.678,168.499,78.786,167.448
C01691=1012.552,-50.321,-110.659,168.465,78.743,167.408
C01692=1012.553,-50.555,-110.639,168.430,78.701,167.369
C01693=1012.553,-50.789,-110.619,168.397,78.659,167.330
C01694=1012.554,-51.022,-110.599,168.362,78.617,167.291
C01695=1012.554,-51.256,-110.579,168.327,78.574,167.251
C01696=1012.555,-51.490,-110.560,168.296,78.531,167.214
C01697=1012.555,-51.723,-110.540,168.262,78.487,167.174
C01698=1012.555,-51.957,-110.520,168.227,78.444,167.135
C01699=1012.556,-52.191,-110.501,168.192,78.399,167.095
C01700=1012.557,-52.425,-110.481,168.160,78.355,167.057
C01701=1012.557,-52.659,-110.461,168.126,78.311,167.018
C01702=1012.558,-52.892,-110.441,168.095,78.267,166.981
C01703=1012.558,-53.126,-110.422,168.061,78.222,166.942
C01704=1012.558,-53.360,-110.401,168.027,78.176,166.902
C01705=1012.558,-53.593,-110.383,167.995,78.131,166.865
C01706=1012.559,-53.827,-110.363,167.962,78.085,166.826
C01707=1012.559,-54.061,-110.343,167.931,78.040,166.789
C01708=1012.560,-54.295,-110.323,167.898,77.994,166.751
C01709=1012.561,-54.529,-110.304,167.866,77.948,166.713
C01710=1012.561,-54.762,-110.283,167.833,77.900,166.674
C01711=1012.562,-54.996,-110.264,167.801,77.854,166.637
C01712=1012.562,-55.230,-110.244,167.769,77.807,166.599
C01713=1012.563,-55.463,-110.224,167.737,77.759,166.561
C01714=1012.563,-55.697,-110.205,167.707,77.711,166.524
C01715=1012.563,-55.931,-110.185,167.673,77.663,166.485
C01716=1012.564,-56.165,-110.166,167.644,77.615,166.449
C01717=1012.564,-56.398,-110.145,167.612,77.566,166.411
C01718=1012.566,-56.632,-110.125,167.581,77.518,166.374
C01719=1012.566,-56.867,-110.105,167.548,77.468,166.336
C01720=1012.566,-57.101,-110.086,167.517,77.419,166.299
C01721=1012.567,-57.335,-110.066,167.487,77.369,166.262
C01722=1012.568,-57.570,-110.047,167.456,77.319,166.225
C01723=1012.569,-57.805,-110.027,167.426,77.269,166.188
C01724=1012.569,-58.039,-110.007,167.396,77.219,166.152
C01725=1012.569,-58.275,-109.987,167.366,77.167,166.115
C01726=1012.570,-58.510,-109.967,167.334,77.116,166.078
C01727=1012.570,-58.746,-109.947,167.305,77.065,166.041
C01728=1012.571,-58.981,-109.928,167.276,77.013,166.005
C01729=1012.572,-59.217,-109.908,167.245,76.961,165.968
C01730=1012.572,-59.453,-109.887,167.215,76.908,165.932
C01731=1012.573,-59.689,-109.867,167.185,76.856,165.895
C01732=1012.574,-59.926,-109.847,167.155,76.802,165.858
C01733=1012.574,-60.162,-109.827,167.126,76.749,165.823
C01734=1012.575,-60.399,-109.807,167.098,76.695,165.787
C01735=1012.575,-60.636,-109.787,167.068,76.642,165.751
C01736=1012.576,-60.873,-109.768,167.039,76.587,165.714
C01737=1012.576,-61.109,-109.747,167.011,76.533,165.679
C01738=1012.577,-61.347,-109.727,166.982,76.478,165.643
C01739=1012.577,-61.585,-109.707,166.955,76.422,165.608
C01740=1012.578,-61.823,-109.686,166.924,76.366,165.571
C01741=1012.578,-62.061,-109.667,166.898,76.311,165.536
C01742=1012.579,-62.299,-109.646,166.869,76.254,165.501
C01743=1012.580,-62.621,-109.619,166.832,76.179,165.453
C01744=1012.582,-63.015,-109.586,166.786,76.083,165.394
C01745=1012.582,-63.254,-109.565,166.757,76.026,165.359
C01746=1012.582,-63.492,-109.546,166.731,75.968,165.324
C01747=1012.584,-63.732,-109.525,166.705,75.910,165.290
C01748=1012.585,-63.971,-109.505,166.676,75.852,165.255
C01749=1012.585,-64.211,-109.485,166.650,75.793,165.220
C01750=1012.586,-64.450,-109.465,166.624,75.734,165.186
C01751=1012.586,-64.690,-109.445,166.596,75.674,165.151
C01752=1012.588,-64.929,-109.424,166.570,75.614,165.116
C01753=1012.588,-65.169,-109.404,166.543,75.554,165.082
C01754=1012.588,-65.409,-109.383,166.518,75.494,165.048
C01755=1012.589,-65.649,-109.362,166.492,75.433,165.013
C01756=1012.590,-65.889,-109.343,166.465,75.372,164.979
C01757=1012.591,-66.129,-109.322,166.441,75.310,164.946
C01758=1012.591,-66.370,-109.302,166.415,75.249,164.912
C01759=1012.592,-66.610,-109.281,166.390,75.187,164.878
C01760=1012.593,-66.850,-109.262,166.365,75.125,164.844
C01761=1012.594,-67.090,-109.241,166.340,75.062,164.811
C01762=1012.595,-67.331,-109.220,166.313,74.999,164.776
C01763=1012.595,-67.572,-109.200,166.291,74.936,164.744
C01764=1012.596,-67.812,-109.179,166.267,74.873,164.711
C01765=1012.597,-68.053,-109.159,166.241,74.808,164.677
C01766=1012.598,-68.295,-109.139,166.218,74.745,164.645
C01767=1012.598,-68.534,-109.118,166.193,74.680,164.611
C01768=1012.600,-68.775,-109.098,166.170,74.616,164.579
C01769=1012.600,-69.017,-109.077,166.147,74.551,164.547
C01770=1012.601,-69.257,-109.057,166.123,74.485,164.514
C01771=1012.602,-69.497,-109.037,166.100,74.419,164.481
C01772=1012.602,-69.739,-109.016,166.077,74.354,164.449
C01773=1012.604,-69.980,-108.996,166.055,74.288,164.418
C01774=1012.605,-70.220,-108.975,166.032,74.221,164.385
C01775=1012.605,-70.461,-108.955,166.010,74.154,164.353
C01776=1012.606,-70.702,-108.935,165.988,74.087,164.322
C01777=1012.607,-70.942,-108.914,165.964,74.019,164.289
C01778=1012.608,-71.182,-108.894,165.943,73.952,164.258
C01779=1012.609,-71.424,-108.873,165.920,73.884,164.226
